LIN {X 0,Y 158.301,Z 763.526,A -85,B 0,C 180,E1 -23831.897,E2 -23831.897} C_VEL
LIN {X 0,Y 156.241,Z 763.233,A -85,B 0,C 180,E1 -23837.005,E2 -23837.005} C_VEL
LIN {X 0,Y 155.491,Z 761.615,A -85,B 0,C 180,E1 -23842.209,E2 -23842.209} C_VEL
LIN {X 0,Y 155.56,Z 760.273,A -85,B 0,C 180,E1 -23844.818,E2 -23844.818} C_VEL
LIN {X 0,Y 155.979,Z 757.524,A -85,B 0,C 180,E1 -23848.711,E2 -23848.711} C_VEL
LIN {X 0,Y 156.074,Z 755.027,A -85,B 0,C 180,E1 -23851.292,E2 -23851.292} C_VEL
LIN {X 0,Y 156.073,Z 750.262,A -85,B 0,C 180,E1 -23855.169,E2 -23855.169} C_VEL
LIN {X 0,Y 156.218,Z 744.142,A -85,B 0,C 180,E1 -23859.06,E2 -23859.06} C_VEL
LIN {X 0,Y 156.866,Z 736.53,A -85,B 0,C 180,E1 -23862.947,E2 -23862.947} C_VEL
LIN {X 0,Y 157.853,Z 728.748,A -85,B 0,C 180,E1 -23866.159,E2 -23866.159} C_VEL
LIN {X 0,Y 159.467,Z 718.303,A -85,B 0,C 180,E1 -23869.638,E2 -23869.638} C_VEL
LIN {X 0,Y 160.165,Z 713.944,A -85,B 0,C 180,E1 -23870.878,E2 -23870.878} C_VEL
LIN {X 0,Y 160.339,Z 710.911,A -85,B 0,C 180,E1 -23871.762,E2 -23871.762} C_VEL
LIN {X 0,Y 159.896,Z 708.03,A -85,B 0,C 180,E1 -23872.707,E2 -23872.707} C_VEL
LIN {X 0,Y 158.002,Z 702.633,A -85,B 0,C 180,E1 -23874.702,E2 -23874.702} C_VEL
LIN {X 0,Y 155.669,Z 695.881,A -85,B 0,C 180,E1 -23877.298,E2 -23877.298} C_VEL
LIN {X 0,Y 155.435,Z 691.449,A -85,B 0,C 180,E1 -23878.779,E2 -23878.779} C_VEL
LIN {X 0,Y 156.41,Z 680.785,A -85,B 0,C 180,E1 -23881.753,E2 -23881.753} C_VEL
LIN {X 0,Y 157.105,Z 669.304,A -85,B 0,C 180,E1 -23884.389,E2 -23884.389} C_VEL
LIN {X 0,Y 157.289,Z 656.551,A -85,B 0,C 180,E1 -23886.771,E2 -23886.771} C_VEL
LIN {X 0,Y 156.753,Z 643.83,A -85,B 0,C 180,E1 -23888.709,E2 -23888.709} C_VEL
LIN {X 0,Y 155.505,Z 632.193,A -85,B 0,C 180,E1 -23890.2,E2 -23890.2} C_VEL
LIN {X 0,Y 154.129,Z 625.609,A -85,B 0,C 180,E1 -23891.054,E2 -23891.054} C_VEL
LIN {X 0,Y 153.301,Z 621.385,A -85,B 0,C 180,E1 -23894.885,E2 -23894.885} C_VEL
LIN {X 0,Y 152.123,Z 615.089,A -85,B 0,C 180,E1 -23900.97,E2 -23900.97} C_VEL
LIN {X 0,Y 151.226,Z 610.219,A -85,B 0,C 180,E1 -23906.103,E2 -23906.103} C_VEL
LIN {X 0,Y 150.323,Z 606.285,A -85,B 0,C 180,E1 -23910.599,E2 -23910.599} C_VEL
LIN {X 0,Y 150.215,Z 605.775,A -85,B 0,C 180,E1 -23911.342,E2 -23911.342} C_VEL
LIN {X 0,Y 150.233,Z 605.772,A -85,B 0,C 180,E1 -23915.099,E2 -23915.099} C_VEL
LIN {X 0,Y 150.374,Z 605.756,A -85,B 0,C 180,E1 -23920.903,E2 -23920.903} C_VEL
LIN {X 0,Y 150.471,Z 605.745,A -85,B 0,C 180,E1 -23926.494,E2 -23926.494} C_VEL
LIN {X 0,Y 150.696,Z 605.716,A -85,B 0,C 180,E1 -23929.248,E2 -23929.248} C_VEL
LIN {X 0,Y 150.769,Z 605.703,A -85,B 0,C 180,E1 -23931.96,E2 -23931.96} C_VEL
LIN {X 0,Y 151.224,Z 605.648,A -85,B 0,C 180,E1 -23939.999,E2 -23939.999} C_VEL
LIN {X 0,Y 150.75,Z 605.699,A -85,B 0,C 180,E1 -23948.039,E2 -23948.039} C_VEL
LIN {X 0,Y 150.62,Z 605.721,A -85,B 0,C 180,E1 -23951.505,E2 -23951.505} C_VEL
LIN {X 0,Y 150.371,Z 605.729,A -85,B 0,C 180,E1 -23956.285,E2 -23956.285} C_VEL
LIN {X 0,Y 150.356,Z 605.756,A -85,B 0,C 180,E1 -23960.791,E2 -23960.791} C_VEL
LIN {X 0,Y 150.249,Z 605.748,A -85,B 0,C 180,E1 -23967.281,E2 -23967.281} C_VEL
LIN {X 0,Y 150.224,Z 605.771,A -85,B 0,C 180,E1 -23972.633,E2 -23972.633} C_VEL
LIN {X 0,Y 150.176,Z 605.777,A -85,B 0,C 180,E1 -23977.471,E2 -23977.471} C_VEL
LIN {X 0,Y 150.153,Z 605.779,A -85,B 0,C 180,E1 -23981.503,E2 -23981.503} C_VEL
LIN {X 0,Y 150.144,Z 605.764,A -85,B 0,C 180,E1 -23985.399,E2 -23985.399} C_VEL
LIN {X 0,Y 150.162,Z 605.778,A -85,B 0,C 180,E1 -23989.06,E2 -23989.06} C_VEL
LIN {X 0,Y 150.218,Z 605.759,A -85,B 0,C 180,E1 -23992.687,E2 -23992.687} C_VEL
LIN {X 0,Y 150.219,Z 605.765,A -85,B 0,C 180,E1 -23997.364,E2 -23997.364} C_VEL
LIN {X 0,Y 150.294,Z 605.761,A -85,B 0,C 180,E1 -24003.948,E2 -24003.948} C_VEL
LIN {X 0,Y 151.357,Z 608.655,A -85,B 0,C 180,E1 -24004.641,E2 -24004.641} C_VEL
LIN {X 0,Y 156.151,Z 618.519,A -85,B 0,C 180,E1 -24007.498,E2 -24007.498} C_VEL
LIN {X 0,Y 159.415,Z 627.15,A -85,B 0,C 180,E1 -24010.001,E2 -24010.001} C_VEL
LIN {X 0,Y 162.002,Z 635.852,A -85,B 0,C 180,E1 -24012.629,E2 -24012.629} C_VEL
LIN {X 0,Y 163.752,Z 643.431,A -85,B 0,C 180,E1 -24015.075,E2 -24015.075} C_VEL
LIN {X 0,Y 161.104,Z 653.934,A -85,B 0,C 180,E1 -24018.039,E2 -24018.039} C_VEL
LIN {X 0,Y 158.728,Z 662.491,A -85,B 0,C 180,E1 -24021.083,E2 -24021.083} C_VEL
LIN {X 0,Y 156.32,Z 670.812,A -85,B 0,C 180,E1 -24024.839,E2 -24024.839} C_VEL
LIN {X 0,Y 154.304,Z 677.372,A -85,B 0,C 180,E1 -24028.562,E2 -24028.562} C_VEL
LIN {X 0,Y 152.679,Z 683.001,A -85,B 0,C 180,E1 -24032.636,E2 -24032.636} C_VEL
LIN {X 0,Y 151.64,Z 687.263,A -85,B 0,C 180,E1 -24036.651,E2 -24036.651} C_VEL
LIN {X 0,Y 151.203,Z 690.46,A -85,B 0,C 180,E1 -24040.712,E2 -24040.712} C_VEL
LIN {X 0,Y 151.19,Z 692.074,A -85,B 0,C 180,E1 -24043.437,E2 -24043.437} C_VEL
LIN {X 0,Y 151.427,Z 693.228,A -85,B 0,C 180,E1 -24046.166,E2 -24046.166} C_VEL
LIN {X 0,Y 152.738,Z 694.356,A -85,B 0,C 180,E1 -24051.596,E2 -24051.596} C_VEL
LIN {X 0,Y 153.787,Z 694.304,A -85,B 0,C 180,E1 -24054.283,E2 -24054.283} C_VEL
LIN {X 0,Y 155.07,Z 693.827,A -85,B 0,C 180,E1 -24056.947,E2 -24056.947} C_VEL
LIN {X 0,Y 156.658,Z 692.946,A -85,B 0,C 180,E1 -24059.567,E2 -24059.567} C_VEL
LIN {X 0,Y 159.152,Z 691.108,A -85,B 0,C 180,E1 -24062.965,E2 -24062.965} C_VEL
LIN {X 0,Y 162.943,Z 687.635,A -85,B 0,C 180,E1 -24067.142,E2 -24067.142} C_VEL
LIN {X 0,Y 166.847,Z 683.387,A -85,B 0,C 180,E1 -24070.696,E2 -24070.696} C_VEL
LIN {X 0,Y 169.613,Z 680.051,A -85,B 0,C 180,E1 -24072.876,E2 -24072.876} C_VEL
LIN {X 0,Y 169.655,Z 678.661,A -85,B 0,C 180,E1 -24074.075,E2 -24074.075} C_VEL
LIN {X 0,Y 160.365,Z 677.774,A -85,B 0,C 180,E1 -24078.901,E2 -24078.901} C_VEL
LIN {X 0,Y 156.701,Z 676.883,A -85,B 0,C 180,E1 -24081.518,E2 -24081.518} C_VEL
LIN {X 0,Y 156.522,Z 676.909,A -85,B 0,C 180,E1 -24081.773,E2 -24081.773} C_VEL
LIN {X 0,Y 154.558,Z 688.668,A -85,B 0,C 180,E1 -24084.33,E2 -24084.33} C_VEL
LIN {X 0,Y 152.548,Z 700.573,A -85,B 0,C 180,E1 -24087.619,E2 -24087.619} C_VEL
LIN {X 0,Y 150.917,Z 709.743,A -85,B 0,C 180,E1 -24090.728,E2 -24090.728} C_VEL
LIN {X 0,Y 149.6,Z 718.707,A -85,B 0,C 180,E1 -24094.423,E2 -24094.423} C_VEL
LIN {X 0,Y 148.6,Z 726.73,A -85,B 0,C 180,E1 -24098.499,E2 -24098.499} C_VEL
LIN {X 0,Y 148.01,Z 733.166,A -85,B 0,C 180,E1 -24102.538,E2 -24102.538} C_VEL
LIN {X 0,Y 147.744,Z 739.641,A -85,B 0,C 180,E1 -24107.641,E2 -24107.641} C_VEL
LIN {X 0,Y 148.22,Z 743.771,A -85,B 0,C 180,E1 -24111.823,E2 -24111.823} C_VEL
LIN {X 0,Y 149.77,Z 747.73,A -85,B 0,C 180,E1 -24117.311,E2 -24117.311} C_VEL
LIN {X 0,Y 152.483,Z 750.261,A -85,B 0,C 180,E1 -24122.643,E2 -24122.643} C_VEL
LIN {X 0,Y 156.515,Z 751.332,A -85,B 0,C 180,E1 -24127.743,E2 -24127.743} C_VEL
LIN {X 0,Y 161.797,Z 751.029,A -85,B 0,C 180,E1 -24132.545,E2 -24132.545} C_VEL
LIN {X 0,Y 168.358,Z 749.378,A -85,B 0,C 180,E1 -24136.991,E2 -24136.991} C_VEL
LIN {X 0,Y 175.968,Z 746.261,A -85,B 0,C 180,E1 -24141.067,E2 -24141.067} C_VEL
LIN {X 0,Y 184.615,Z 741.664,A -85,B 0,C 180,E1 -24144.757,E2 -24144.757} C_VEL
LIN {X 0,Y 194.158,Z 735.354,A -85,B 0,C 180,E1 -24148.072,E2 -24148.072} C_VEL
LIN {X 0,Y 203.161,Z 728.262,A -85,B 0,C 180,E1 -24150.681,E2 -24150.681} C_VEL
LIN {X 0,Y 205.743,Z 726,A -85,B 0,C 180,E1 -24151.357,E2 -24151.357} C_VEL
LIN {X 0,Y 208.061,Z 723.711,A -85,B 0,C 180,E1 -24152.716,E2 -24152.716} C_VEL
LIN {X 0,Y 209.401,Z 722.346,A -85,B 0,C 180,E1 -24153.628,E2 -24153.628} C_VEL
LIN {X 0,Y 210.467,Z 721.212,A -85,B 0,C 180,E1 -24154.589,E2 -24154.589} C_VEL
LIN {X 0,Y 211.809,Z 720.065,A -85,B 0,C 180,E1 -24157.221,E2 -24157.221} C_VEL
LIN {X 0,Y 212.367,Z 720.043,A -85,B 0,C 180,E1 -24158.961,E2 -24158.961} C_VEL
LIN {X 0,Y 209.953,Z 722.891,A -85,B 0,C 180,E1 -24160.353,E2 -24160.353} C_VEL
LIN {X 0,Y 204.984,Z 728.502,A -85,B 0,C 180,E1 -24162.515,E2 -24162.515} C_VEL
LIN {X 0,Y 199.025,Z 734.248,A -85,B 0,C 180,E1 -24164.354,E2 -24164.354} C_VEL
LIN {X 0,Y 190.597,Z 741.609,A -85,B 0,C 180,E1 -24166.99,E2 -24166.99} C_VEL
LIN {X 0,Y 181.392,Z 748.549,A -85,B 0,C 180,E1 -24170.264,E2 -24170.264} C_VEL
LIN {X 0,Y 174.835,Z 752.856,A -85,B 0,C 180,E1 -24172.92,E2 -24172.92} C_VEL
LIN {X 0,Y 167.216,Z 757.285,A -85,B 0,C 180,E1 -24176.884,E2 -24176.884} C_VEL
LIN {X 0,Y 160.578,Z 760.437,A -85,B 0,C 180,E1 -24181.224,E2 -24181.224} C_VEL
LIN {X 0,Y 155.447,Z 762.353,A -85,B 0,C 180,E1 -24185.992,E2 -24185.992} C_VEL
LIN {X 0,Y 151.563,Z 763.014,A -85,B 0,C 180,E1 -24191.062,E2 -24191.062} C_VEL
LIN {X 0,Y 149.342,Z 762.396,A -85,B 0,C 180,E1 -24196.393,E2 -24196.393} C_VEL
LIN {X 0,Y 148.515,Z 760.499,A -85,B 0,C 180,E1 -24201.841,E2 -24201.841} C_VEL
LIN {X 0,Y 148.602,Z 759.026,A -85,B 0,C 180,E1 -24204.575,E2 -24204.575} C_VEL
LIN {X 0,Y 149.043,Z 756.066,A -85,B 0,C 180,E1 -24208.652,E2 -24208.652} C_VEL
LIN {X 0,Y 149.112,Z 753.462,A -85,B 0,C 180,E1 -24211.353,E2 -24211.353} C_VEL
LIN {X 0,Y 149.116,Z 748.437,A -85,B 0,C 180,E1 -24215.411,E2 -24215.411} C_VEL
LIN {X 0,Y 149.329,Z 742.021,A -85,B 0,C 180,E1 -24219.482,E2 -24219.482} C_VEL
LIN {X 0,Y 150.05,Z 733.972,A -85,B 0,C 180,E1 -24223.546,E2 -24223.546} C_VEL
LIN {X 0,Y 151.356,Z 724.046,A -85,B 0,C 180,E1 -24227.569,E2 -24227.569} C_VEL
LIN {X 0,Y 153.223,Z 712.726,A -85,B 0,C 180,E1 -24231.177,E2 -24231.177} C_VEL
LIN {X 0,Y 153.805,Z 709.196,A -85,B 0,C 180,E1 -24232.149,E2 -24232.149} C_VEL
LIN {X 0,Y 154.545,Z 700.824,A -85,B 0,C 180,E1 -24235.597,E2 -24235.597} C_VEL
LIN {X 0,Y 155.435,Z 691.449,A -85,B 0,C 180,E1 -24238.779,E2 -24238.779} C_VEL
LIN {X 0,Y 155.253,Z 686.965,A -85,B 0,C 180,E1 -24240.18,E2 -24240.18} C_VEL
LIN {X 0,Y 153.152,Z 679.582,A -85,B 0,C 180,E1 -24242.533,E2 -24242.533} C_VEL
LIN {X 0,Y 151.003,Z 671.94,A -85,B 0,C 180,E1 -24244.804,E2 -24244.804} C_VEL
LIN {X 0,Y 150.63,Z 666.943,A -85,B 0,C 180,E1 -24246.014,E2 -24246.014} C_VEL
LIN {X 0,Y 150.901,Z 653.621,A -85,B 0,C 180,E1 -24248.535,E2 -24248.535} C_VEL
LIN {X 0,Y 150.259,Z 639.839,A -85,B 0,C 180,E1 -24250.68,E2 -24250.68} C_VEL
LIN {X 0,Y 148.895,Z 630.887,A -85,B 0,C 180,E1 -24251.953,E2 -24251.953} C_VEL
LIN {X 0,Y 148.126,Z 628.352,A -85,B 0,C 180,E1 -24252.388,E2 -24252.388} C_VEL
LIN {X 0,Y 146.693,Z 624.312,A -85,B 0,C 180,E1 -24253.127,E2 -24253.127} C_VEL
LIN {X 0,Y 145.429,Z 618.159,A -85,B 0,C 180,E1 -24259.278,E2 -24259.278} C_VEL
LIN {X 0,Y 144.594,Z 613.43,A -85,B 0,C 180,E1 -24264.318,E2 -24264.318} C_VEL
LIN {X 0,Y 143.805,Z 609.245,A -85,B 0,C 180,E1 -24269.125,E2 -24269.125} C_VEL
LIN {X 0,Y 143.216,Z 606.645,A -85,B 0,C 180,E1 -24272.488,E2 -24272.488} C_VEL
LIN {X 0,Y 143.284,Z 606.64,A -85,B 0,C 180,E1 -24278.745,E2 -24278.745} C_VEL
LIN {X 0,Y 143.323,Z 606.636,A -85,B 0,C 180,E1 -24282.888,E2 -24282.888} C_VEL
LIN {X 0,Y 143.609,Z 606.598,A -85,B 0,C 180,E1 -24288.71,E2 -24288.71} C_VEL
LIN {X 0,Y 143.691,Z 606.585,A -85,B 0,C 180,E1 -24291.561,E2 -24291.561} C_VEL
LIN {X 0,Y 144.183,Z 606.525,A -85,B 0,C 180,E1 -24299.999,E2 -24299.999} C_VEL
LIN {X 0,Y 143.671,Z 606.583,A -85,B 0,C 180,E1 -24308.438,E2 -24308.438} C_VEL
LIN {X 0,Y 143.553,Z 606.602,A -85,B 0,C 180,E1 -24311.711,E2 -24311.711} C_VEL
LIN {X 0,Y 143.309,Z 606.611,A -85,B 0,C 180,E1 -24317.111,E2 -24317.111} C_VEL
LIN {X 0,Y 143.282,Z 606.637,A -85,B 0,C 180,E1 -24321.253,E2 -24321.253} C_VEL
LIN {X 0,Y 143.196,Z 606.629,A -85,B 0,C 180,E1 -24327.936,E2 -24327.936} C_VEL
LIN {X 0,Y 143.151,Z 606.65,A -85,B 0,C 180,E1 -24333.42,E2 -24333.42} C_VEL
LIN {X 0,Y 143.064,Z 606.661,A -85,B 0,C 180,E1 -24339.688,E2 -24339.688} C_VEL
LIN {X 0,Y 143.064,Z 606.651,A -85,B 0,C 180,E1 -24343.451,E2 -24343.451} C_VEL
LIN {X 0,Y 143.075,Z 606.658,A -85,B 0,C 180,E1 -24347.459,E2 -24347.459} C_VEL
LIN {X 0,Y 143.11,Z 606.644,A -85,B 0,C 180,E1 -24351.788,E2 -24351.788} C_VEL
LIN {X 0,Y 143.187,Z 606.641,A -85,B 0,C 180,E1 -24357.32,E2 -24357.32} C_VEL
LIN {X 0,Y 143.193,Z 606.812,A -85,B 0,C 180,E1 -24361.958,E2 -24361.958} C_VEL
LIN {X 0,Y 144.278,Z 609.57,A -85,B 0,C 180,E1 -24362.706,E2 -24362.706} C_VEL
LIN {X 0,Y 145.183,Z 610.769,A -85,B 0,C 180,E1 -24363.162,E2 -24363.162} C_VEL
LIN {X 0,Y 150.317,Z 621.884,A -85,B 0,C 180,E1 -24366.646,E2 -24366.646} C_VEL
LIN {X 0,Y 153.24,Z 629.925,A -85,B 0,C 180,E1 -24369.159,E2 -24369.159} C_VEL
LIN {X 0,Y 155.662,Z 638.385,A -85,B 0,C 180,E1 -24371.911,E2 -24371.911} C_VEL
LIN {X 0,Y 157.084,Z 644.663,A -85,B 0,C 180,E1 -24374.091,E2 -24374.091} C_VEL
LIN {X 0,Y 156.799,Z 646.889,A -85,B 0,C 180,E1 -24374.73,E2 -24374.73} C_VEL
LIN {X 0,Y 154.248,Z 656.012,A -85,B 0,C 180,E1 -24377.499,E2 -24377.499} C_VEL
LIN {X 0,Y 151.293,Z 665.84,A -85,B 0,C 180,E1 -24381.314,E2 -24381.314} C_VEL
LIN {X 0,Y 149.248,Z 672.533,A -85,B 0,C 180,E1 -24384.593,E2 -24384.593} C_VEL
LIN {X 0,Y 147.198,Z 678.965,A -85,B 0,C 180,E1 -24388.493,E2 -24388.493} C_VEL
LIN {X 0,Y 145.543,Z 684.488,A -85,B 0,C 180,E1 -24392.765,E2 -24392.765} C_VEL
LIN {X 0,Y 144.535,Z 688.645,A -85,B 0,C 180,E1 -24396.98,E2 -24396.98} C_VEL
LIN {X 0,Y 144.119,Z 692.599,A -85,B 0,C 180,E1 -24402.765,E2 -24402.765} C_VEL
LIN {X 0,Y 144.507,Z 694.378,A -85,B 0,C 180,E1 -24406.963,E2 -24406.963} C_VEL
LIN {X 0,Y 145.122,Z 695.092,A -85,B 0,C 180,E1 -24409.813,E2 -24409.813} C_VEL
LIN {X 0,Y 146.778,Z 695.372,A -85,B 0,C 180,E1 -24414.531,E2 -24414.531} C_VEL
LIN {X 0,Y 148.63,Z 694.749,A -85,B 0,C 180,E1 -24418.217,E2 -24418.217} C_VEL
LIN {X 0,Y 150.388,Z 693.823,A -85,B 0,C 180,E1 -24420.931,E2 -24420.931} C_VEL
LIN {X 0,Y 152.794,Z 692.109,A -85,B 0,C 180,E1 -24424.114,E2 -24424.114} C_VEL
LIN {X 0,Y 157.18,Z 688.318,A -85,B 0,C 180,E1 -24428.751,E2 -24428.751} C_VEL
LIN {X 0,Y 161.717,Z 683.57,A -85,B 0,C 180,E1 -24432.653,E2 -24432.653} C_VEL
LIN {X 0,Y 162.855,Z 682.122,A -85,B 0,C 180,E1 -24433.665,E2 -24433.665} C_VEL
LIN {X 0,Y 148.855,Z 680.705,A -85,B 0,C 180,E1 -24442.138,E2 -24442.138} C_VEL
LIN {X 0,Y 148.753,Z 680.967,A -85,B 0,C 180,E1 -24442.302,E2 -24442.302} C_VEL
LIN {X 0,Y 146.676,Z 693.215,A -85,B 0,C 180,E1 -24445.321,E2 -24445.321} C_VEL
LIN {X 0,Y 144.857,Z 703.701,A -85,B 0,C 180,E1 -24448.565,E2 -24448.565} C_VEL
LIN {X 0,Y 143.193,Z 713.525,A -85,B 0,C 180,E1 -24452.326,E2 -24452.326} C_VEL
LIN {X 0,Y 141.938,Z 722.688,A -85,B 0,C 180,E1 -24456.666,E2 -24456.666} C_VEL
LIN {X 0,Y 141.116,Z 730.253,A -85,B 0,C 180,E1 -24461.121,E2 -24461.121} C_VEL
LIN {X 0,Y 140.701,Z 736.342,A -85,B 0,C 180,E1 -24465.538,E2 -24465.538} C_VEL
LIN {X 0,Y 140.859,Z 741.194,A -85,B 0,C 180,E1 -24469.944,E2 -24469.944} C_VEL
LIN {X 0,Y 141.708,Z 745.045,A -85,B 0,C 180,E1 -24474.309,E2 -24474.309} C_VEL
LIN {X 0,Y 143.696,Z 748.787,A -85,B 0,C 180,E1 -24480.001,E2 -24480.001} C_VEL
LIN {X 0,Y 147.161,Z 751.048,A -85,B 0,C 180,E1 -24485.482,E2 -24485.482} C_VEL
LIN {X 0,Y 151.908,Z 751.944,A -85,B 0,C 180,E1 -24490.666,E2 -24490.666} C_VEL
LIN {X 0,Y 157.986,Z 751.504,A -85,B 0,C 180,E1 -24495.481,E2 -24495.481} C_VEL
LIN {X 0,Y 165.278,Z 749.664,A -85,B 0,C 180,E1 -24499.889,E2 -24499.889} C_VEL
LIN {X 0,Y 173.654,Z 746.42,A -85,B 0,C 180,E1 -24503.874,E2 -24503.874} C_VEL
LIN {X 0,Y 183.018,Z 741.682,A -85,B 0,C 180,E1 -24507.44,E2 -24507.44} C_VEL
LIN {X 0,Y 193.229,Z 735.201,A -85,B 0,C 180,E1 -24510.611,E2 -24510.611} C_VEL
LIN {X 0,Y 201.391,Z 729.127,A -85,B 0,C 180,E1 -24512.745,E2 -24512.745} C_VEL
LIN {X 0,Y 204.235,Z 726.638,A -85,B 0,C 180,E1 -24514.327,E2 -24514.327} C_VEL
LIN {X 0,Y 205.566,Z 725.568,A -85,B 0,C 180,E1 -24515.536,E2 -24515.536} C_VEL
LIN {X 0,Y 206.692,Z 724.829,A -85,B 0,C 180,E1 -24517.738,E2 -24517.738} C_VEL
LIN {X 0,Y 206.7,Z 725.081,A -85,B 0,C 180,E1 -24518.557,E2 -24518.557} C_VEL
LIN {X 0,Y 202.724,Z 729.061,A -85,B 0,C 180,E1 -24520.301,E2 -24520.301} C_VEL
LIN {X 0,Y 199.389,Z 732.222,A -85,B 0,C 180,E1 -24521.498,E2 -24521.498} C_VEL
LIN {X 0,Y 190.514,Z 739.613,A -85,B 0,C 180,E1 -24524.002,E2 -24524.002} C_VEL
LIN {X 0,Y 180.858,Z 746.721,A -85,B 0,C 180,E1 -24527.157,E2 -24527.157} C_VEL
LIN {X 0,Y 171.462,Z 752.467,A -85,B 0,C 180,E1 -24530.559,E2 -24530.559} C_VEL
LIN {X 0,Y 165.169,Z 755.88,A -85,B 0,C 180,E1 -24533.44,E2 -24533.44} C_VEL
LIN {X 0,Y 157.666,Z 759.265,A -85,B 0,C 180,E1 -24537.666,E2 -24537.666} C_VEL
LIN {X 0,Y 151.555,Z 761.417,A -85,B 0,C 180,E1 -24542.375,E2 -24542.375} C_VEL
LIN {X 0,Y 146.794,Z 762.358,A -85,B 0,C 180,E1 -24547.482,E2 -24547.482} C_VEL
LIN {X 0,Y 143.448,Z 762.076,A -85,B 0,C 180,E1 -24552.908,E2 -24552.908} C_VEL
LIN {X 0,Y 141.816,Z 760.568,A -85,B 0,C 180,E1 -24558.569,E2 -24558.569} C_VEL
LIN {X 0,Y 141.655,Z 757.737,A -85,B 0,C 180,E1 -24564.308,E2 -24564.308} C_VEL
LIN {X 0,Y 142.121,Z 754.561,A -85,B 0,C 180,E1 -24568.586,E2 -24568.586} C_VEL
LIN {X 0,Y 142.183,Z 751.749,A -85,B 0,C 180,E1 -24571.419,E2 -24571.419} C_VEL
LIN {X 0,Y 142.16,Z 746.462,A -85,B 0,C 180,E1 -24575.677,E2 -24575.677} C_VEL
LIN {X 0,Y 142.412,Z 739.746,A -85,B 0,C 180,E1 -24579.947,E2 -24579.947} C_VEL
LIN {X 0,Y 143.232,Z 731.342,A -85,B 0,C 180,E1 -24584.204,E2 -24584.204} C_VEL
LIN {X 0,Y 144.669,Z 720.828,A -85,B 0,C 180,E1 -24588.41,E2 -24588.41} C_VEL
LIN {X 0,Y 146.443,Z 710.42,A -85,B 0,C 180,E1 -24591.837,E2 -24591.837} C_VEL
LIN {X 0,Y 147.102,Z 706.091,A -85,B 0,C 180,E1 -24593.883,E2 -24593.883} C_VEL
LIN {X 0,Y 147.974,Z 697.037,A -85,B 0,C 180,E1 -24597.588,E2 -24597.588} C_VEL
LIN {X 0,Y 149.049,Z 687.304,A -85,B 0,C 180,E1 -24600.852,E2 -24600.852} C_VEL
LIN {X 0,Y 150.078,Z 676.231,A -85,B 0,C 180,E1 -24603.88,E2 -24603.88} C_VEL
LIN {X 0,Y 150.63,Z 666.943,A -85,B 0,C 180,E1 -24606.014,E2 -24606.014} C_VEL
LIN {X 0,Y 150.216,Z 661.901,A -85,B 0,C 180,E1 -24607.18,E2 -24607.18} C_VEL
LIN {X 0,Y 147.668,Z 653.919,A -85,B 0,C 180,E1 -24609.236,E2 -24609.236} C_VEL
LIN {X 0,Y 144.9,Z 645.742,A -85,B 0,C 180,E1 -24611.2,E2 -24611.2} C_VEL
LIN {X 0,Y 144.081,Z 640.381,A -85,B 0,C 180,E1 -24612.168,E2 -24612.168} C_VEL
LIN {X 0,Y 142.976,Z 632.465,A -85,B 0,C 180,E1 -24613.424,E2 -24613.424} C_VEL
LIN {X 0,Y 140.902,Z 627.616,A -85,B 0,C 180,E1 -24614.503,E2 -24614.503} C_VEL
LIN {X 0,Y 139.436,Z 624.264,A -85,B 0,C 180,E1 -24615.233,E2 -24615.233} C_VEL
LIN {X 0,Y 139.138,Z 623.031,A -85,B 0,C 180,E1 -24615.504,E2 -24615.504} C_VEL
LIN {X 0,Y 138.198,Z 617.877,A -85,B 0,C 180,E1 -24620.98,E2 -24620.98} C_VEL
LIN {X 0,Y 137.446,Z 613.695,A -85,B 0,C 180,E1 -24625.772,E2 -24625.772} C_VEL
LIN {X 0,Y 136.912,Z 610.962,A -85,B 0,C 180,E1 -24629.113,E2 -24629.113} C_VEL
LIN {X 0,Y 136.135,Z 607.528,A -85,B 0,C 180,E1 -24633.764,E2 -24633.764} C_VEL
LIN {X 0,Y 136.251,Z 607.517,A -85,B 0,C 180,E1 -24638.833,E2 -24638.833} C_VEL
LIN {X 0,Y 136.292,Z 607.512,A -85,B 0,C 180,E1 -24645.058,E2 -24645.058} C_VEL
LIN {X 0,Y 136.508,Z 607.481,A -85,B 0,C 180,E1 -24648.114,E2 -24648.114} C_VEL
LIN {X 0,Y 136.615,Z 607.468,A -85,B 0,C 180,E1 -24651.121,E2 -24651.121} C_VEL
LIN {X 0,Y 137.14,Z 607.402,A -85,B 0,C 180,E1 -24659.999,E2 -24659.999} C_VEL
LIN {X 0,Y 136.598,Z 607.466,A -85,B 0,C 180,E1 -24668.878,E2 -24668.878} C_VEL
LIN {X 0,Y 136.497,Z 607.479,A -85,B 0,C 180,E1 -24671.953,E2 -24671.953} C_VEL
LIN {X 0,Y 136.249,Z 607.496,A -85,B 0,C 180,E1 -24678.027,E2 -24678.027} C_VEL
LIN {X 0,Y 136.203,Z 607.519,A -85,B 0,C 180,E1 -24681.747,E2 -24681.747} C_VEL
LIN {X 0,Y 136.122,Z 607.514,A -85,B 0,C 180,E1 -24688.628,E2 -24688.628} C_VEL
LIN {X 0,Y 136.048,Z 607.534,A -85,B 0,C 180,E1 -24694.626,E2 -24694.626} C_VEL
LIN {X 0,Y 136.034,Z 607.535,A -85,B 0,C 180,E1 -24699.196,E2 -24699.196} C_VEL
LIN {X 0,Y 136.005,Z 607.528,A -85,B 0,C 180,E1 -24703.657,E2 -24703.657} C_VEL
LIN {X 0,Y 136.038,Z 607.535,A -85,B 0,C 180,E1 -24707.806,E2 -24707.806} C_VEL
LIN {X 0,Y 136.059,Z 607.522,A -85,B 0,C 180,E1 -24711.692,E2 -24711.692} C_VEL
LIN {X 0,Y 136.092,Z 607.532,A -85,B 0,C 180,E1 -24715.715,E2 -24715.715} C_VEL
LIN {X 0,Y 136.084,Z 607.644,A -85,B 0,C 180,E1 -24719.661,E2 -24719.661} C_VEL
LIN {X 0,Y 137.091,Z 610.383,A -85,B 0,C 180,E1 -24720.456,E2 -24720.456} C_VEL
LIN {X 0,Y 140.441,Z 616.118,A -85,B 0,C 180,E1 -24722.591,E2 -24722.591} C_VEL
LIN {X 0,Y 144.604,Z 625.56,A -85,B 0,C 180,E1 -24725.832,E2 -24725.832} C_VEL
LIN {X 0,Y 147.586,Z 634.312,A -85,B 0,C 180,E1 -24728.832,E2 -24728.832} C_VEL
LIN {X 0,Y 149.727,Z 642.745,A -85,B 0,C 180,E1 -24731.825,E2 -24731.825} C_VEL
LIN {X 0,Y 150.595,Z 646.913,A -85,B 0,C 180,E1 -24733.386,E2 -24733.386} C_VEL
LIN {X 0,Y 147.916,Z 656.228,A -85,B 0,C 180,E1 -24736.255,E2 -24736.255} C_VEL
LIN {X 0,Y 145.289,Z 664.727,A -85,B 0,C 180,E1 -24739.546,E2 -24739.546} C_VEL
LIN {X 0,Y 142.6,Z 673.013,A -85,B 0,C 180,E1 -24743.631,E2 -24743.631} C_VEL
LIN {X 0,Y 140.354,Z 679.742,A -85,B 0,C 180,E1 -24747.845,E2 -24747.845} C_VEL
LIN {X 0,Y 138.394,Z 685.947,A -85,B 0,C 180,E1 -24752.908,E2 -24752.908} C_VEL
LIN {X 0,Y 137.44,Z 689.992,A -85,B 0,C 180,E1 -24757.342,E2 -24757.342} C_VEL
LIN {X 0,Y 137.089,Z 693.663,A -85,B 0,C 180,E1 -24763.087,E2 -24763.087} C_VEL
LIN {X 0,Y 137.614,Z 695.528,A -85,B 0,C 180,E1 -24767.841,E2 -24767.841} C_VEL
LIN {X 0,Y 138.336,Z 696.197,A -85,B 0,C 180,E1 -24770.829,E2 -24770.829} C_VEL
LIN {X 0,Y 140.04,Z 696.395,A -85,B 0,C 180,E1 -24775.402,E2 -24775.402} C_VEL
LIN {X 0,Y 142.271,Z 695.674,A -85,B 0,C 180,E1 -24779.6,E2 -24779.6} C_VEL
LIN {X 0,Y 144.183,Z 694.68,A -85,B 0,C 180,E1 -24782.42,E2 -24782.42} C_VEL
LIN {X 0,Y 146.535,Z 693.096,A -85,B 0,C 180,E1 -24785.381,E2 -24785.381} C_VEL
LIN {X 0,Y 150.163,Z 690.2,A -85,B 0,C 180,E1 -24789.182,E2 -24789.182} C_VEL
LIN {X 0,Y 155.275,Z 685.304,A -85,B 0,C 180,E1 -24793.601,E2 -24793.601} C_VEL
LIN {X 0,Y 144.04,Z 684.497,A -85,B 0,C 180,E1 -24800.634,E2 -24800.634} C_VEL
LIN {X 0,Y 141.905,Z 684.676,A -85,B 0,C 180,E1 -24801.755,E2 -24801.755} C_VEL
LIN {X 0,Y 141.096,Z 684.436,A -85,B 0,C 180,E1 -24802.804,E2 -24802.804} C_VEL
LIN {X 0,Y 138.98,Z 696.61,A -85,B 0,C 180,E1 -24806.204,E2 -24806.204} C_VEL
LIN {X 0,Y 137.088,Z 706.873,A -85,B 0,C 180,E1 -24809.768,E2 -24809.768} C_VEL
LIN {X 0,Y 135.638,Z 716.443,A -85,B 0,C 180,E1 -24813.871,E2 -24813.871} C_VEL
LIN {X 0,Y 134.49,Z 725.292,A -85,B 0,C 180,E1 -24818.545,E2 -24818.545} C_VEL
LIN {X 0,Y 133.863,Z 732.394,A -85,B 0,C 180,E1 -24823.218,E2 -24823.218} C_VEL
LIN {X 0,Y 133.673,Z 738.074,A -85,B 0,C 180,E1 -24827.861,E2 -24827.861} C_VEL
LIN {X 0,Y 134.517,Z 743.974,A -85,B 0,C 180,E1 -24834.003,E2 -24834.003} C_VEL
LIN {X 0,Y 136.485,Z 748.19,A -85,B 0,C 180,E1 -24840.001,E2 -24840.001} C_VEL
LIN {X 0,Y 139.963,Z 750.948,A -85,B 0,C 180,E1 -24845.765,E2 -24845.765} C_VEL
LIN {X 0,Y 144.81,Z 752.354,A -85,B 0,C 180,E1 -24851.195,E2 -24851.195} C_VEL
LIN {X 0,Y 151.072,Z 752.429,A -85,B 0,C 180,E1 -24856.209,E2 -24856.209} C_VEL
LIN {X 0,Y 158.573,Z 751.131,A -85,B 0,C 180,E1 -24860.768,E2 -24860.768} C_VEL
LIN {X 0,Y 167.186,Z 748.485,A -85,B 0,C 180,E1 -24864.859,E2 -24864.859} C_VEL
LIN {X 0,Y 176.772,Z 744.391,A -85,B 0,C 180,E1 -24868.497,E2 -24868.497} C_VEL
LIN {X 0,Y 187.272,Z 738.671,A -85,B 0,C 180,E1 -24871.696,E2 -24871.696} C_VEL
LIN {X 0,Y 195.29,Z 733.406,A -85,B 0,C 180,E1 -24873.771,E2 -24873.771} C_VEL
LIN {X 0,Y 198.065,Z 731.426,A -85,B 0,C 180,E1 -24874.593,E2 -24874.593} C_VEL
LIN {X 0,Y 200.307,Z 729.872,A -85,B 0,C 180,E1 -24876.202,E2 -24876.202} C_VEL
LIN {X 0,Y 200.488,Z 729.775,A -85,B 0,C 180,E1 -24876.58,E2 -24876.58} C_VEL
LIN {X 0,Y 200.502,Z 730.053,A -85,B 0,C 180,E1 -24878.097,E2 -24878.097} C_VEL
LIN {X 0,Y 196.281,Z 733.704,A -85,B 0,C 180,E1 -24879.665,E2 -24879.665} C_VEL
LIN {X 0,Y 185.812,Z 741.561,A -85,B 0,C 180,E1 -24882.48,E2 -24882.48} C_VEL
LIN {X 0,Y 175.8,Z 748.064,A -85,B 0,C 180,E1 -24885.608,E2 -24885.608} C_VEL
LIN {X 0,Y 166.1,Z 753.373,A -85,B 0,C 180,E1 -24889.02,E2 -24889.02} C_VEL
LIN {X 0,Y 159.544,Z 756.397,A -85,B 0,C 180,E1 -24891.927,E2 -24891.927} C_VEL
LIN {X 0,Y 151.716,Z 759.409,A -85,B 0,C 180,E1 -24896.232,E2 -24896.232} C_VEL
LIN {X 0,Y 145.278,Z 761.216,A -85,B 0,C 180,E1 -24901.072,E2 -24901.072} C_VEL
LIN {X 0,Y 140.262,Z 761.823,A -85,B 0,C 180,E1 -24906.372,E2 -24906.372} C_VEL
LIN {X 0,Y 136.706,Z 761.207,A -85,B 0,C 180,E1 -24912.037,E2 -24912.037} C_VEL
LIN {X 0,Y 134.921,Z 759.41,A -85,B 0,C 180,E1 -24917.977,E2 -24917.977} C_VEL
LIN {X 0,Y 134.716,Z 756.283,A -85,B 0,C 180,E1 -24924.014,E2 -24924.014} C_VEL
LIN {X 0,Y 135.223,Z 752.931,A -85,B 0,C 180,E1 -24928.514,E2 -24928.514} C_VEL
LIN {X 0,Y 135.244,Z 749.965,A -85,B 0,C 180,E1 -24931.492,E2 -24931.492} C_VEL
LIN {X 0,Y 135.215,Z 744.365,A -85,B 0,C 180,E1 -24935.97,E2 -24935.97} C_VEL
LIN {X 0,Y 135.492,Z 737.534,A -85,B 0,C 180,E1 -24940.311,E2 -24940.311} C_VEL
LIN {X 0,Y 136.419,Z 728.462,A -85,B 0,C 180,E1 -24944.93,E2 -24944.93} C_VEL
LIN {X 0,Y 137.698,Z 719.529,A -85,B 0,C 180,E1 -24948.605,E2 -24948.605} C_VEL
LIN {X 0,Y 138.968,Z 712.174,A -85,B 0,C 180,E1 -24951.123,E2 -24951.123} C_VEL
LIN {X 0,Y 140.001,Z 707.36,A -85,B 0,C 180,E1 -24953.681,E2 -24953.681} C_VEL
LIN {X 0,Y 140.829,Z 698.981,A -85,B 0,C 180,E1 -24957.494,E2 -24957.494} C_VEL
LIN {X 0,Y 142.116,Z 688.696,A -85,B 0,C 180,E1 -24961.285,E2 -24961.285} C_VEL
LIN {X 0,Y 143.418,Z 677.065,A -85,B 0,C 180,E1 -24964.759,E2 -24964.759} C_VEL
LIN {X 0,Y 144.186,Z 666.571,A -85,B 0,C 180,E1 -24967.34,E2 -24967.34} C_VEL
LIN {X 0,Y 144.607,Z 653.809,A -85,B 0,C 180,E1 -24969.907,E2 -24969.907} C_VEL
LIN {X 0,Y 144.081,Z 640.381,A -85,B 0,C 180,E1 -24972.168,E2 -24972.168} C_VEL
LIN {X 0,Y 143.19,Z 637.035,A -85,B 0,C 180,E1 -24972.854,E2 -24972.854} C_VEL
LIN {X 0,Y 141.323,Z 634.287,A -85,B 0,C 180,E1 -24973.717,E2 -24973.717} C_VEL
LIN {X 0,Y 134.057,Z 627.235,A -85,B 0,C 180,E1 -24976.741,E2 -24976.741} C_VEL
LIN {X 0,Y 133.391,Z 626.284,A -85,B 0,C 180,E1 -24977.072,E2 -24977.072} C_VEL
LIN {X 0,Y 131.883,Z 622.815,A -85,B 0,C 180,E1 -24977.928,E2 -24977.928} C_VEL
LIN {X 0,Y 131.627,Z 621.631,A -85,B 0,C 180,E1 -24978.245,E2 -24978.245} C_VEL
LIN {X 0,Y 130.838,Z 616.899,A -85,B 0,C 180,E1 -24983.78,E2 -24983.78} C_VEL
LIN {X 0,Y 130.049,Z 612.749,A -85,B 0,C 180,E1 -24988.984,E2 -24988.984} C_VEL
LIN {X 0,Y 129.067,Z 608.409,A -85,B 0,C 180,E1 -24995.145,E2 -24995.145} C_VEL
LIN {X 0,Y 129.167,Z 608.397,A -85,B 0,C 180,E1 -25000.945,E2 -25000.945} C_VEL
LIN {X 0,Y 129.425,Z 608.363,A -85,B 0,C 180,E1 -25007.815,E2 -25007.815} C_VEL
LIN {X 0,Y 129.537,Z 608.351,A -85,B 0,C 180,E1 -25010.631,E2 -25010.631} C_VEL
LIN {X 0,Y 130.095,Z 608.279,A -85,B 0,C 180,E1 -25019.999,E2 -25019.999} C_VEL
LIN {X 0,Y 129.523,Z 608.349,A -85,B 0,C 180,E1 -25029.367,E2 -25029.367} C_VEL
LIN {X 0,Y 129.398,Z 608.359,A -85,B 0,C 180,E1 -25032.546,E2 -25032.546} C_VEL
LIN {X 0,Y 129.16,Z 608.386,A -85,B 0,C 180,E1 -25039.054,E2 -25039.054} C_VEL
LIN {X 0,Y 129.113,Z 608.401,A -85,B 0,C 180,E1 -25042.396,E2 -25042.396} C_VEL
LIN {X 0,Y 129.04,Z 608.401,A -85,B 0,C 180,E1 -25049.371,E2 -25049.371} C_VEL
LIN {X 0,Y 128.964,Z 608.419,A -85,B 0,C 180,E1 -25055.166,E2 -25055.166} C_VEL
LIN {X 0,Y 128.947,Z 608.422,A -85,B 0,C 180,E1 -25060.845,E2 -25060.845} C_VEL
LIN {X 0,Y 128.928,Z 608.405,A -85,B 0,C 180,E1 -25065.123,E2 -25065.123} C_VEL
LIN {X 0,Y 128.984,Z 608.414,A -85,B 0,C 180,E1 -25069.712,E2 -25069.712} C_VEL
LIN {X 0,Y 128.994,Z 608.415,A -85,B 0,C 180,E1 -25074.808,E2 -25074.808} C_VEL
LIN {X 0,Y 129.012,Z 608.497,A -85,B 0,C 180,E1 -25077.063,E2 -25077.063} C_VEL
LIN {X 0,Y 129.97,Z 611.191,A -85,B 0,C 180,E1 -25077.926,E2 -25077.926} C_VEL
LIN {X 0,Y 131.399,Z 613.232,A -85,B 0,C 180,E1 -25078.843,E2 -25078.843} C_VEL
LIN {X 0,Y 135.884,Z 621.939,A -85,B 0,C 180,E1 -25082.256,E2 -25082.256} C_VEL
LIN {X 0,Y 139.694,Z 631.464,A -85,B 0,C 180,E1 -25085.826,E2 -25085.826} C_VEL
LIN {X 0,Y 142.302,Z 640.294,A -85,B 0,C 180,E1 -25089.141,E2 -25089.141} C_VEL
LIN {X 0,Y 143.911,Z 647.899,A -85,B 0,C 180,E1 -25092.122,E2 -25092.122} C_VEL
LIN {X 0,Y 143.957,Z 649.074,A -85,B 0,C 180,E1 -25092.547,E2 -25092.547} C_VEL
LIN {X 0,Y 141.092,Z 658.286,A -85,B 0,C 180,E1 -25095.576,E2 -25095.576} C_VEL
LIN {X 0,Y 138.335,Z 666.589,A -85,B 0,C 180,E1 -25099.014,E2 -25099.014} C_VEL
LIN {X 0,Y 135.56,Z 674.732,A -85,B 0,C 180,E1 -25103.299,E2 -25103.299} C_VEL
LIN {X 0,Y 133.581,Z 680.319,A -85,B 0,C 180,E1 -25106.981,E2 -25106.981} C_VEL
LIN {X 0,Y 131.745,Z 685.81,A -85,B 0,C 180,E1 -25111.526,E2 -25111.526} C_VEL
LIN {X 0,Y 130.571,Z 690.126,A -85,B 0,C 180,E1 -25116.177,E2 -25116.177} C_VEL
LIN {X 0,Y 130.146,Z 692.438,A -85,B 0,C 180,E1 -25119.32,E2 -25119.32} C_VEL
LIN {X 0,Y 130.077,Z 694.737,A -85,B 0,C 180,E1 -25123.465,E2 -25123.465} C_VEL
LIN {X 0,Y 130.775,Z 696.678,A -85,B 0,C 180,E1 -25128.808,E2 -25128.808} C_VEL
LIN {X 0,Y 131.589,Z 697.272,A -85,B 0,C 180,E1 -25131.951,E2 -25131.951} C_VEL
LIN {X 0,Y 134.213,Z 697.216,A -85,B 0,C 180,E1 -25138.114,E2 -25138.114} C_VEL
LIN {X 0,Y 136,Z 696.595,A -85,B 0,C 180,E1 -25141.112,E2 -25141.112} C_VEL
LIN {X 0,Y 140.344,Z 694.087,A -85,B 0,C 180,E1 -25146.754,E2 -25146.754} C_VEL
LIN {X 0,Y 144.57,Z 690.883,A -85,B 0,C 180,E1 -25151.013,E2 -25151.013} C_VEL
LIN {X 0,Y 146.066,Z 689.601,A -85,B 0,C 180,E1 -25152.343,E2 -25152.343} C_VEL
LIN {X 0,Y 146.665,Z 688.289,A -85,B 0,C 180,E1 -25154.048,E2 -25154.048} C_VEL
LIN {X 0,Y 139.208,Z 687.938,A -85,B 0,C 180,E1 -25158.982,E2 -25158.982} C_VEL
LIN {X 0,Y 136.323,Z 688.103,A -85,B 0,C 180,E1 -25160.647,E2 -25160.647} C_VEL
LIN {X 0,Y 133.709,Z 687.921,A -85,B 0,C 180,E1 -25162.823,E2 -25162.823} C_VEL
LIN {X 0,Y 133.417,Z 687.69,A -85,B 0,C 180,E1 -25163.432,E2 -25163.432} C_VEL
LIN {X 0,Y 131.258,Z 699.683,A -85,B 0,C 180,E1 -25167.173,E2 -25167.173} C_VEL
LIN {X 0,Y 129.264,Z 710.952,A -85,B 0,C 180,E1 -25171.594,E2 -25171.594} C_VEL
LIN {X 0,Y 128.069,Z 719.396,A -85,B 0,C 180,E1 -25175.698,E2 -25175.698} C_VEL
LIN {X 0,Y 127.151,Z 727.618,A -85,B 0,C 180,E1 -25180.633,E2 -25180.633} C_VEL
LIN {X 0,Y 126.652,Z 734.258,A -85,B 0,C 180,E1 -25185.541,E2 -25185.541} C_VEL
LIN {X 0,Y 126.804,Z 739.66,A -85,B 0,C 180,E1 -25190.43,E2 -25190.43} C_VEL
LIN {X 0,Y 128.172,Z 745.231,A -85,B 0,C 180,E1 -25196.858,E2 -25196.858} C_VEL
LIN {X 0,Y 130.843,Z 749.191,A -85,B 0,C 180,E1 -25203.08,E2 -25203.08} C_VEL
LIN {X 0,Y 135.242,Z 751.824,A -85,B 0,C 180,E1 -25209.141,E2 -25209.141} C_VEL
LIN {X 0,Y 140.743,Z 753.038,A -85,B 0,C 180,E1 -25214.459,E2 -25214.459} C_VEL
LIN {X 0,Y 147.874,Z 752.94,A -85,B 0,C 180,E1 -25219.433,E2 -25219.433} C_VEL
LIN {X 0,Y 156.145,Z 751.544,A -85,B 0,C 180,E1 -25223.898,E2 -25223.898} C_VEL
LIN {X 0,Y 165.557,Z 748.793,A -85,B 0,C 180,E1 -25227.838,E2 -25227.838} C_VEL
LIN {X 0,Y 175.847,Z 744.583,A -85,B 0,C 180,E1 -25231.304,E2 -25231.304} C_VEL
LIN {X 0,Y 187.456,Z 738.489,A -85,B 0,C 180,E1 -25234.435,E2 -25234.435} C_VEL
LIN {X 0,Y 192.701,Z 735.258,A -85,B 0,C 180,E1 -25235.701,E2 -25235.701} C_VEL
LIN {X 0,Y 194.452,Z 734.274,A -85,B 0,C 180,E1 -25237.336,E2 -25237.336} C_VEL
LIN {X 0,Y 192.059,Z 736.097,A -85,B 0,C 180,E1 -25238.121,E2 -25238.121} C_VEL
LIN {X 0,Y 181.239,Z 743.373,A -85,B 0,C 180,E1 -25240.877,E2 -25240.877} C_VEL
LIN {X 0,Y 170.869,Z 749.366,A -85,B 0,C 180,E1 -25243.967,E2 -25243.967} C_VEL
LIN {X 0,Y 160.835,Z 754.131,A -85,B 0,C 180,E1 -25247.37,E2 -25247.37} C_VEL
LIN {X 0,Y 154.047,Z 756.862,A -85,B 0,C 180,E1 -25250.308,E2 -25250.308} C_VEL
LIN {X 0,Y 145.874,Z 759.449,A -85,B 0,C 180,E1 -25254.683,E2 -25254.683} C_VEL
LIN {X 0,Y 139.104,Z 760.879,A -85,B 0,C 180,E1 -25259.657,E2 -25259.657} C_VEL
LIN {X 0,Y 133.79,Z 761.154,A -85,B 0,C 180,E1 -25265.154,E2 -25265.154} C_VEL
LIN {X 0,Y 129.999,Z 760.262,A -85,B 0,C 180,E1 -25271.076,E2 -25271.076} C_VEL
LIN {X 0,Y 128.052,Z 758.163,A -85,B 0,C 180,E1 -25277.321,E2 -25277.321} C_VEL
LIN {X 0,Y 127.801,Z 754.755,A -85,B 0,C 180,E1 -25283.689,E2 -25283.689} C_VEL
LIN {X 0,Y 128.331,Z 751.174,A -85,B 0,C 180,E1 -25288.434,E2 -25288.434} C_VEL
LIN {X 0,Y 128.325,Z 748.02,A -85,B 0,C 180,E1 -25291.572,E2 -25291.572} C_VEL
LIN {X 0,Y 128.289,Z 742.133,A -85,B 0,C 180,E1 -25296.293,E2 -25296.293} C_VEL
LIN {X 0,Y 128.648,Z 734.937,A -85,B 0,C 180,E1 -25300.866,E2 -25300.866} C_VEL
LIN {X 0,Y 129.453,Z 727.073,A -85,B 0,C 180,E1 -25304.947,E2 -25304.947} C_VEL
LIN {X 0,Y 130.964,Z 716.948,A -85,B 0,C 180,E1 -25309.192,E2 -25309.192} C_VEL
LIN {X 0,Y 131.635,Z 713.136,A -85,B 0,C 180,E1 -25310.717,E2 -25310.717} C_VEL
LIN {X 0,Y 132.966,Z 707.133,A -85,B 0,C 180,E1 -25314.184,E2 -25314.184} C_VEL
LIN {X 0,Y 133.902,Z 698.93,A -85,B 0,C 180,E1 -25318.191,E2 -25318.191} C_VEL
LIN {X 0,Y 135.334,Z 688.93,A -85,B 0,C 180,E1 -25322.163,E2 -25322.163} C_VEL
LIN {X 0,Y 136.791,Z 677.66,A -85,B 0,C 180,E1 -25325.765,E2 -25325.765} C_VEL
LIN {X 0,Y 137.897,Z 665.226,A -85,B 0,C 180,E1 -25329.011,E2 -25329.011} C_VEL
LIN {X 0,Y 138.404,Z 653.153,A -85,B 0,C 180,E1 -25331.555,E2 -25331.555} C_VEL
LIN {X 0,Y 137.965,Z 639.86,A -85,B 0,C 180,E1 -25333.936,E2 -25333.936} C_VEL
LIN {X 0,Y 137.261,Z 635.377,A -85,B 0,C 180,E1 -25334.758,E2 -25334.758} C_VEL
LIN {X 0,Y 135.432,Z 630.909,A -85,B 0,C 180,E1 -25335.889,E2 -25335.889} C_VEL
LIN {X 0,Y 133.629,Z 626.672,A -85,B 0,C 180,E1 -25336.948,E2 -25336.948} C_VEL
LIN {X 0,Y 133.391,Z 626.284,A -85,B 0,C 180,E1 -25337.072,E2 -25337.072} C_VEL
LIN {X 0,Y 131.327,Z 623.807,A -85,B 0,C 180,E1 -25338.123,E2 -25338.123} C_VEL
LIN {X 0,Y 127.538,Z 621.015,A -85,B 0,C 180,E1 -25340.279,E2 -25340.279} C_VEL
LIN {X 0,Y 124.554,Z 618.993,A -85,B 0,C 180,E1 -25342.898,E2 -25342.898} C_VEL
LIN {X 0,Y 123.755,Z 617.732,A -85,B 0,C 180,E1 -25344.637,E2 -25344.637} C_VEL
LIN {X 0,Y 123.149,Z 614.38,A -85,B 0,C 180,E1 -25349.093,E2 -25349.093} C_VEL
LIN {X 0,Y 122.279,Z 610.678,A -85,B 0,C 180,E1 -25354.463,E2 -25354.463} C_VEL
LIN {X 0,Y 122.03,Z 609.285,A -85,B 0,C 180,E1 -25356.857,E2 -25356.857} C_VEL
LIN {X 0,Y 122.125,Z 609.276,A -85,B 0,C 180,E1 -25363.276,E2 -25363.276} C_VEL
LIN {X 0,Y 122.372,Z 609.242,A -85,B 0,C 180,E1 -25367.522,E2 -25367.522} C_VEL
LIN {X 0,Y 122.463,Z 609.234,A -85,B 0,C 180,E1 -25370.085,E2 -25370.085} C_VEL
LIN {X 0,Y 122.615,Z 609.207,A -85,B 0,C 180,E1 -25376.713,E2 -25376.713} C_VEL
LIN {X 0,Y 123.049,Z 609.156,A -85,B 0,C 180,E1 -25379.999,E2 -25379.999} C_VEL
LIN {X 0,Y 122.421,Z 609.213,A -85,B 0,C 180,E1 -25387.184,E2 -25387.184} C_VEL
LIN {X 0,Y 122.369,Z 609.235,A -85,B 0,C 180,E1 -25392.471,E2 -25392.471} C_VEL
LIN {X 0,Y 122.051,Z 609.279,A -85,B 0,C 180,E1 -25400.211,E2 -25400.211} C_VEL
LIN {X 0,Y 121.988,Z 609.28,A -85,B 0,C 180,E1 -25403.782,E2 -25403.782} C_VEL
LIN {X 0,Y 121.943,Z 609.291,A -85,B 0,C 180,E1 -25410.169,E2 -25410.169} C_VEL
LIN {X 0,Y 121.888,Z 609.302,A -85,B 0,C 180,E1 -25416.169,E2 -25416.169} C_VEL
LIN {X 0,Y 121.883,Z 609.301,A -85,B 0,C 180,E1 -25421.44,E2 -25421.44} C_VEL
LIN {X 0,Y 121.905,Z 609.298,A -85,B 0,C 180,E1 -25428.542,E2 -25428.542} C_VEL
LIN {X 0,Y 121.959,Z 609.404,A -85,B 0,C 180,E1 -25434.053,E2 -25434.053} C_VEL
LIN {X 0,Y 122.894,Z 612.032,A -85,B 0,C 180,E1 -25435.005,E2 -25435.005} C_VEL
LIN {X 0,Y 126.36,Z 617.595,A -85,B 0,C 180,E1 -25437.687,E2 -25437.687} C_VEL
LIN {X 0,Y 130.661,Z 626.397,A -85,B 0,C 180,E1 -25441.473,E2 -25441.473} C_VEL
LIN {X 0,Y 133.708,Z 634.497,A -85,B 0,C 180,E1 -25444.781,E2 -25444.781} C_VEL
LIN {X 0,Y 136.118,Z 643.199,A -85,B 0,C 180,E1 -25448.333,E2 -25448.333} C_VEL
LIN {X 0,Y 137.426,Z 649.896,A -85,B 0,C 180,E1 -25451.145,E2 -25451.145} C_VEL
LIN {X 0,Y 136.505,Z 653.596,A -85,B 0,C 180,E1 -25452.391,E2 -25452.391} C_VEL
LIN {X 0,Y 133.66,Z 662.087,A -85,B 0,C 180,E1 -25455.534,E2 -25455.534} C_VEL
LIN {X 0,Y 130.928,Z 669.919,A -85,B 0,C 180,E1 -25459.168,E2 -25459.168} C_VEL
LIN {X 0,Y 128.042,Z 677.624,A -85,B 0,C 180,E1 -25463.695,E2 -25463.695} C_VEL
LIN {X 0,Y 125.785,Z 683.837,A -85,B 0,C 180,E1 -25468.396,E2 -25468.396} C_VEL
LIN {X 0,Y 124.132,Z 688.81,A -85,B 0,C 180,E1 -25473.243,E2 -25473.243} C_VEL
LIN {X 0,Y 123.22,Z 692.662,A -85,B 0,C 180,E1 -25478.195,E2 -25478.195} C_VEL
LIN {X 0,Y 123.06,Z 695.804,A -85,B 0,C 180,E1 -25483.867,E2 -25483.867} C_VEL
LIN {X 0,Y 123.948,Z 697.818,A -85,B 0,C 180,E1 -25489.886,E2 -25489.886} C_VEL
LIN {X 0,Y 126.232,Z 698.452,A -85,B 0,C 180,E1 -25496.446,E2 -25496.446} C_VEL
LIN {X 0,Y 127.859,Z 698.186,A -85,B 0,C 180,E1 -25499.646,E2 -25499.646} C_VEL
LIN {X 0,Y 129.829,Z 697.481,A -85,B 0,C 180,E1 -25502.77,E2 -25502.77} C_VEL
LIN {X 0,Y 134.284,Z 695.06,A -85,B 0,C 180,E1 -25508.277,E2 -25508.277} C_VEL
LIN {X 0,Y 138.816,Z 691.817,A -85,B 0,C 180,E1 -25512.698,E2 -25512.698} C_VEL
LIN {X 0,Y 139.11,Z 691.07,A -85,B 0,C 180,E1 -25513.918,E2 -25513.918} C_VEL
LIN {X 0,Y 134.329,Z 691.007,A -85,B 0,C 180,E1 -25517.146,E2 -25517.146} C_VEL
LIN {X 0,Y 130.353,Z 691.206,A -85,B 0,C 180,E1 -25519.687,E2 -25519.687} C_VEL
LIN {X 0,Y 126.993,Z 691.131,A -85,B 0,C 180,E1 -25522.502,E2 -25522.502} C_VEL
LIN {X 0,Y 125.696,Z 690.884,A -85,B 0,C 180,E1 -25524.175,E2 -25524.175} C_VEL
LIN {X 0,Y 123.529,Z 702.72,A -85,B 0,C 180,E1 -25528.345,E2 -25528.345} C_VEL
LIN {X 0,Y 121.894,Z 712.34,A -85,B 0,C 180,E1 -25532.534,E2 -25532.534} C_VEL
LIN {X 0,Y 120.584,Z 722.278,A -85,B 0,C 180,E1 -25537.92,E2 -25537.92} C_VEL
LIN {X 0,Y 119.861,Z 729.792,A -85,B 0,C 180,E1 -25542.953,E2 -25542.953} C_VEL
LIN {X 0,Y 119.66,Z 736.033,A -85,B 0,C 180,E1 -25548.139,E2 -25548.139} C_VEL
LIN {X 0,Y 120.234,Z 741.345,A -85,B 0,C 180,E1 -25553.533,E2 -25553.533} C_VEL
LIN {X 0,Y 122.098,Z 746.373,A -85,B 0,C 180,E1 -25560.001,E2 -25560.001} C_VEL
LIN {X 0,Y 125.594,Z 750.132,A -85,B 0,C 180,E1 -25566.427,E2 -25566.427} C_VEL
LIN {X 0,Y 130.672,Z 752.571,A -85,B 0,C 180,E1 -25572.425,E2 -25572.425} C_VEL
LIN {X 0,Y 137.245,Z 753.67,A -85,B 0,C 180,E1 -25577.895,E2 -25577.895} C_VEL
LIN {X 0,Y 145.187,Z 753.472,A -85,B 0,C 180,E1 -25582.785,E2 -25582.785} C_VEL
LIN {X 0,Y 154.314,Z 751.975,A -85,B 0,C 180,E1 -25587.094,E2 -25587.094} C_VEL
LIN {X 0,Y 164.411,Z 749.158,A -85,B 0,C 180,E1 -25590.862,E2 -25590.862} C_VEL
LIN {X 0,Y 175.436,Z 744.824,A -85,B 0,C 180,E1 -25594.115,E2 -25594.115} C_VEL
LIN {X 0,Y 186.218,Z 739.465,A -85,B 0,C 180,E1 -25596.724,E2 -25596.724} C_VEL
LIN {X 0,Y 185.163,Z 740.13,A -85,B 0,C 180,E1 -25597.153,E2 -25597.153} C_VEL
LIN {X 0,Y 174.061,Z 746.548,A -85,B 0,C 180,E1 -25599.905,E2 -25599.905} C_VEL
LIN {X 0,Y 163.41,Z 751.725,A -85,B 0,C 180,E1 -25603.022,E2 -25603.022} C_VEL
LIN {X 0,Y 153.263,Z 755.704,A -85,B 0,C 180,E1 -25606.545,E2 -25606.545} C_VEL
LIN {X 0,Y 144.301,Z 758.468,A -85,B 0,C 180,E1 -25610.721,E2 -25610.721} C_VEL
LIN {X 0,Y 136.366,Z 760.077,A -85,B 0,C 180,E1 -25615.468,E2 -25615.468} C_VEL
LIN {X 0,Y 129.992,Z 760.567,A -85,B 0,C 180,E1 -25620.887,E2 -25620.887} C_VEL
LIN {X 0,Y 125.092,Z 759.913,A -85,B 0,C 180,E1 -25626.845,E2 -25626.845} C_VEL
LIN {X 0,Y 122.077,Z 758.14,A -85,B 0,C 180,E1 -25633.274,E2 -25633.274} C_VEL
LIN {X 0,Y 120.873,Z 755.12,A -85,B 0,C 180,E1 -25639.958,E2 -25639.958} C_VEL
LIN {X 0,Y 121.034,Z 751.959,A -85,B 0,C 180,E1 -25645.006,E2 -25645.006} C_VEL
LIN {X 0,Y 121.473,Z 749.302,A -85,B 0,C 180,E1 -25648.345,E2 -25648.345} C_VEL
LIN {X 0,Y 121.414,Z 745.966,A -85,B 0,C 180,E1 -25651.662,E2 -25651.662} C_VEL
LIN {X 0,Y 121.389,Z 739.721,A -85,B 0,C 180,E1 -25656.652,E2 -25656.652} C_VEL
LIN {X 0,Y 121.745,Z 732.896,A -85,B 0,C 180,E1 -25661.074,E2 -25661.074} C_VEL
LIN {X 0,Y 122.768,Z 723.922,A -85,B 0,C 180,E1 -25665.782,E2 -25665.782} C_VEL
LIN {X 0,Y 124.193,Z 714.542,A -85,B 0,C 180,E1 -25669.852,E2 -25669.852} C_VEL
LIN {X 0,Y 125.754,Z 708.361,A -85,B 0,C 180,E1 -25673.905,E2 -25673.905} C_VEL
LIN {X 0,Y 126.837,Z 700.1,A -85,B 0,C 180,E1 -25678.371,E2 -25678.371} C_VEL
LIN {X 0,Y 128.425,Z 690.159,A -85,B 0,C 180,E1 -25682.714,E2 -25682.714} C_VEL
LIN {X 0,Y 130.044,Z 679.502,A -85,B 0,C 180,E1 -25686.478,E2 -25686.478} C_VEL
LIN {X 0,Y 131.244,Z 669.145,A -85,B 0,C 180,E1 -25689.49,E2 -25689.49} C_VEL
LIN {X 0,Y 132.126,Z 657.325,A -85,B 0,C 180,E1 -25692.327,E2 -25692.327} C_VEL
LIN {X 0,Y 132.234,Z 644.097,A -85,B 0,C 180,E1 -25694.996,E2 -25694.996} C_VEL
LIN {X 0,Y 131.706,Z 638.611,A -85,B 0,C 180,E1 -25696.075,E2 -25696.075} C_VEL
LIN {X 0,Y 128.402,Z 630.308,A -85,B 0,C 180,E1 -25698.437,E2 -25698.437} C_VEL
LIN {X 0,Y 126.311,Z 625.467,A -85,B 0,C 180,E1 -25699.827,E2 -25699.827} C_VEL
LIN {X 0,Y 124.524,Z 621.647,A -85,B 0,C 180,E1 -25700.974,E2 -25700.974} C_VEL
LIN {X 0,Y 124.22,Z 620.414,A -85,B 0,C 180,E1 -25701.251,E2 -25701.251} C_VEL
LIN {X 0,Y 123.755,Z 617.732,A -85,B 0,C 180,E1 -25704.637,E2 -25704.637} C_VEL
LIN {X 0,Y 122.836,Z 616.595,A -85,B 0,C 180,E1 -25706.335,E2 -25706.335} C_VEL
LIN {X 0,Y 119.658,Z 615.283,A -85,B 0,C 180,E1 -25709.045,E2 -25709.045} C_VEL
LIN {X 0,Y 116.437,Z 613.999,A -85,B 0,C 180,E1 -25711.9,E2 -25711.9} C_VEL
LIN {X 0,Y 115.519,Z 612.946,A -85,B 0,C 180,E1 -25713.773,E2 -25713.773} C_VEL
LIN {X 0,Y 115.003,Z 610.161,A -85,B 0,C 180,E1 -25718.488,E2 -25718.488} C_VEL
LIN {X 0,Y 115.155,Z 610.146,A -85,B 0,C 180,E1 -25725.869,E2 -25725.869} C_VEL
LIN {X 0,Y 115.4,Z 610.114,A -85,B 0,C 180,E1 -25729.471,E2 -25729.471} C_VEL
LIN {X 0,Y 115.541,Z 610.088,A -85,B 0,C 180,E1 -25736.511,E2 -25736.511} C_VEL
LIN {X 0,Y 116.001,Z 610.034,A -85,B 0,C 180,E1 -25739.999,E2 -25739.999} C_VEL
LIN {X 0,Y 115.387,Z 610.091,A -85,B 0,C 180,E1 -25747.087,E2 -25747.087} C_VEL
LIN {X 0,Y 115.29,Z 610.114,A -85,B 0,C 180,E1 -25752.736,E2 -25752.736} C_VEL
LIN {X 0,Y 115.018,Z 610.134,A -85,B 0,C 180,E1 -25757.788,E2 -25757.788} C_VEL
LIN {X 0,Y 114.952,Z 610.158,A -85,B 0,C 180,E1 -25763.49,E2 -25763.49} C_VEL
LIN {X 0,Y 114.866,Z 610.177,A -85,B 0,C 180,E1 -25771.06,E2 -25771.06} C_VEL
LIN {X 0,Y 114.785,Z 610.183,A -85,B 0,C 180,E1 -25777.752,E2 -25777.752} C_VEL
LIN {X 0,Y 114.796,Z 610.174,A -85,B 0,C 180,E1 -25782.717,E2 -25782.717} C_VEL
LIN {X 0,Y 114.847,Z 610.172,A -85,B 0,C 180,E1 -25789.961,E2 -25789.961} C_VEL
LIN {X 0,Y 114.869,Z 610.231,A -85,B 0,C 180,E1 -25790.435,E2 -25790.435} C_VEL
LIN {X 0,Y 115.785,Z 612.961,A -85,B 0,C 180,E1 -25791.538,E2 -25791.538} C_VEL
LIN {X 0,Y 117.156,Z 614.584,A -85,B 0,C 180,E1 -25792.638,E2 -25792.638} C_VEL
LIN {X 0,Y 121.836,Z 623.057,A -85,B 0,C 180,E1 -25796.996,E2 -25796.996} C_VEL
LIN {X 0,Y 125.219,Z 630.332,A -85,B 0,C 180,E1 -25800.447,E2 -25800.447} C_VEL
LIN {X 0,Y 128.272,Z 639.239,A -85,B 0,C 180,E1 -25804.413,E2 -25804.413} C_VEL
LIN {X 0,Y 130.137,Z 646.828,A -85,B 0,C 180,E1 -25807.785,E2 -25807.785} C_VEL
LIN {X 0,Y 130.962,Z 651.851,A -85,B 0,C 180,E1 -25810.074,E2 -25810.074} C_VEL
LIN {X 0,Y 128.133,Z 660.558,A -85,B 0,C 180,E1 -25813.261,E2 -25813.261} C_VEL
LIN {X 0,Y 125.06,Z 668.821,A -85,B 0,C 180,E1 -25817.007,E2 -25817.007} C_VEL
LIN {X 0,Y 121.949,Z 676.933,A -85,B 0,C 180,E1 -25821.713,E2 -25821.713} C_VEL
LIN {X 0,Y 119.375,Z 683.514,A -85,B 0,C 180,E1 -25826.622,E2 -25826.622} C_VEL
LIN {X 0,Y 117.471,Z 688.773,A -85,B 0,C 180,E1 -25831.711,E2 -25831.711} C_VEL
LIN {X 0,Y 116.331,Z 692.883,A -85,B 0,C 180,E1 -25836.937,E2 -25836.937} C_VEL
LIN {X 0,Y 115.999,Z 695.019,A -85,B 0,C 180,E1 -25840.469,E2 -25840.469} C_VEL
LIN {X 0,Y 116.054,Z 696.874,A -85,B 0,C 180,E1 -25844.326,E2 -25844.326} C_VEL
LIN {X 0,Y 116.423,Z 698.056,A -85,B 0,C 180,E1 -25847.564,E2 -25847.564} C_VEL
LIN {X 0,Y 117.186,Z 698.923,A -85,B 0,C 180,E1 -25851.087,E2 -25851.087} C_VEL
LIN {X 0,Y 119.767,Z 699.471,A -85,B 0,C 180,E1 -25857.994,E2 -25857.994} C_VEL
LIN {X 0,Y 121.603,Z 699.14,A -85,B 0,C 180,E1 -25861.339,E2 -25861.339} C_VEL
LIN {X 0,Y 123.773,Z 698.36,A -85,B 0,C 180,E1 -25864.594,E2 -25864.594} C_VEL
LIN {X 0,Y 128.271,Z 696.059,A -85,B 0,C 180,E1 -25869.911,E2 -25869.911} C_VEL
LIN {X 0,Y 130.664,Z 694.556,A -85,B 0,C 180,E1 -25872.243,E2 -25872.243} C_VEL
LIN {X 0,Y 131.427,Z 693.674,A -85,B 0,C 180,E1 -25873.792,E2 -25873.792} C_VEL
LIN {X 0,Y 121.846,Z 694.069,A -85,B 0,C 180,E1 -25880.621,E2 -25880.621} C_VEL
LIN {X 0,Y 118.183,Z 693.956,A -85,B 0,C 180,E1 -25884.565,E2 -25884.565} C_VEL
LIN {X 0,Y 118.018,Z 693.916,A -85,B 0,C 180,E1 -25885.16,E2 -25885.16} C_VEL
LIN {X 0,Y 116.042,Z 704.167,A -85,B 0,C 180,E1 -25889.11,E2 -25889.11} C_VEL
LIN {X 0,Y 114.319,Z 715.341,A -85,B 0,C 180,E1 -25894.512,E2 -25894.512} C_VEL
LIN {X 0,Y 113.394,Z 722.709,A -85,B 0,C 180,E1 -25898.907,E2 -25898.907} C_VEL
LIN {X 0,Y 112.726,Z 730.57,A -85,B 0,C 180,E1 -25904.636,E2 -25904.636} C_VEL
LIN {X 0,Y 112.834,Z 737.608,A -85,B 0,C 180,E1 -25911.043,E2 -25911.043} C_VEL
LIN {X 0,Y 113.842,Z 742.454,A -85,B 0,C 180,E1 -25916.462,E2 -25916.462} C_VEL
LIN {X 0,Y 116.483,Z 747.444,A -85,B 0,C 180,E1 -25923.46,E2 -25923.46} C_VEL
LIN {X 0,Y 120.818,Z 751.045,A -85,B 0,C 180,E1 -25930.051,E2 -25930.051} C_VEL
LIN {X 0,Y 126.799,Z 753.315,A -85,B 0,C 180,E1 -25936.09,E2 -25936.09} C_VEL
LIN {X 0,Y 134.316,Z 754.3,A -85,B 0,C 180,E1 -25941.487,E2 -25941.487} C_VEL
LIN {X 0,Y 143.074,Z 754.019,A -85,B 0,C 180,E1 -25946.239,E2 -25946.239} C_VEL
LIN {X 0,Y 153.021,Z 752.466,A -85,B 0,C 180,E1 -25950.347,E2 -25950.347} C_VEL
LIN {X 0,Y 163.85,Z 749.532,A -85,B 0,C 180,E1 -25953.892,E2 -25953.892} C_VEL
LIN {X 0,Y 173.571,Z 745.967,A -85,B 0,C 180,E1 -25956.456,E2 -25956.456} C_VEL
LIN {X 0,Y 171.895,Z 746.919,A -85,B 0,C 180,E1 -25957.531,E2 -25957.531} C_VEL
LIN {X 0,Y 161.441,Z 751.589,A -85,B 0,C 180,E1 -25960.379,E2 -25960.379} C_VEL
LIN {X 0,Y 153.336,Z 754.532,A -85,B 0,C 180,E1 -25962.836,E2 -25962.836} C_VEL
LIN {X 0,Y 143.421,Z 757.457,A -85,B 0,C 180,E1 -25966.687,E2 -25966.687} C_VEL
LIN {X 0,Y 134.556,Z 759.26,A -85,B 0,C 180,E1 -25971.191,E2 -25971.191} C_VEL
LIN {X 0,Y 127.053,Z 759.953,A -85,B 0,C 180,E1 -25976.42,E2 -25976.42} C_VEL
LIN {X 0,Y 121.095,Z 759.542,A -85,B 0,C 180,E1 -25982.339,E2 -25982.339} C_VEL
LIN {X 0,Y 116.76,Z 757.996,A -85,B 0,C 180,E1 -25988.833,E2 -25988.833} C_VEL
LIN {X 0,Y 114.461,Z 755.312,A -85,B 0,C 180,E1 -25995.786,E2 -25995.786} C_VEL
LIN {X 0,Y 114.087,Z 751.329,A -85,B 0,C 180,E1 -26002.926,E2 -26002.926} C_VEL
LIN {X 0,Y 114.626,Z 747.307,A -85,B 0,C 180,E1 -26008.247,E2 -26008.247} C_VEL
LIN {X 0,Y 114.512,Z 742.801,A -85,B 0,C 180,E1 -26012.641,E2 -26012.641} C_VEL
LIN {X 0,Y 114.572,Z 735.903,A -85,B 0,C 180,E1 -26017.936,E2 -26017.936} C_VEL
LIN {X 0,Y 115.193,Z 727.551,A -85,B 0,C 180,E1 -26023.089,E2 -26023.089} C_VEL
LIN {X 0,Y 116.344,Z 718.602,A -85,B 0,C 180,E1 -26027.583,E2 -26027.583} C_VEL
LIN {X 0,Y 116.788,Z 715.742,A -85,B 0,C 180,E1 -26028.875,E2 -26028.875} C_VEL
LIN {X 0,Y 118.766,Z 708.083,A -85,B 0,C 180,E1 -26034.474,E2 -26034.474} C_VEL
LIN {X 0,Y 119.836,Z 700.661,A -85,B 0,C 180,E1 -26038.843,E2 -26038.843} C_VEL
LIN {X 0,Y 121.522,Z 691.3,A -85,B 0,C 180,E1 -26043.33,E2 -26043.33} C_VEL
LIN {X 0,Y 123.427,Z 680.252,A -85,B 0,C 180,E1 -26047.568,E2 -26047.568} C_VEL
LIN {X 0,Y 125.057,Z 668.172,A -85,B 0,C 180,E1 -26051.329,E2 -26051.329} C_VEL
LIN {X 0,Y 126.061,Z 657.341,A -85,B 0,C 180,E1 -26054.083,E2 -26054.083} C_VEL
LIN {X 0,Y 126.357,Z 644.107,A -85,B 0,C 180,E1 -26056.941,E2 -26056.941} C_VEL
LIN {X 0,Y 126.176,Z 641.768,A -85,B 0,C 180,E1 -26057.462,E2 -26057.462} C_VEL
LIN {X 0,Y 123.216,Z 633.951,A -85,B 0,C 180,E1 -26059.948,E2 -26059.948} C_VEL
LIN {X 0,Y 121.433,Z 629.495,A -85,B 0,C 180,E1 -26061.39,E2 -26061.39} C_VEL
LIN {X 0,Y 119.293,Z 624.543,A -85,B 0,C 180,E1 -26063.041,E2 -26063.041} C_VEL
LIN {X 0,Y 117.282,Z 620.718,A -85,B 0,C 180,E1 -26064.512,E2 -26064.512} C_VEL
LIN {X 0,Y 116.753,Z 618.87,A -85,B 0,C 180,E1 -26065.119,E2 -26065.119} C_VEL
LIN {X 0,Y 115.892,Z 614.778,A -85,B 0,C 180,E1 -26070.977,E2 -26070.977} C_VEL
LIN {X 0,Y 115.519,Z 612.946,A -85,B 0,C 180,E1 -26073.773,E2 -26073.773} C_VEL
LIN {X 0,Y 114.591,Z 611.601,A -85,B 0,C 180,E1 -26076.582,E2 -26076.582} C_VEL
LIN {X 0,Y 112.95,Z 610.945,A -85,B 0,C 180,E1 -26079.428,E2 -26079.428} C_VEL
LIN {X 0,Y 108.609,Z 610.956,A -85,B 0,C 180,E1 -26087.452,E2 -26087.452} C_VEL
LIN {X 0,Y 108.281,Z 610.993,A -85,B 0,C 180,E1 -26089.578,E2 -26089.578} C_VEL
LIN {X 0,Y 108.467,Z 610.969,A -85,B 0,C 180,E1 -26096.284,E2 -26096.284} C_VEL
LIN {X 0,Y 108.951,Z 610.912,A -85,B 0,C 180,E1 -26099.999,E2 -26099.999} C_VEL
LIN {X 0,Y 108.337,Z 610.972,A -85,B 0,C 180,E1 -26107.453,E2 -26107.453} C_VEL
LIN {X 0,Y 108.207,Z 610.992,A -85,B 0,C 180,E1 -26113.018,E2 -26113.018} C_VEL
LIN {X 0,Y 107.91,Z 611.03,A -85,B 0,C 180,E1 -26119.003,E2 -26119.003} C_VEL
LIN {X 0,Y 107.864,Z 611.034,A -85,B 0,C 180,E1 -26124.183,E2 -26124.183} C_VEL
LIN {X 0,Y 107.788,Z 611.059,A -85,B 0,C 180,E1 -26132.04,E2 -26132.04} C_VEL
LIN {X 0,Y 107.694,Z 611.064,A -85,B 0,C 180,E1 -26138.449,E2 -26138.449} C_VEL
LIN {X 0,Y 107.708,Z 611.174,A -85,B 0,C 180,E1 -26145.964,E2 -26145.964} C_VEL
LIN {X 0,Y 108.678,Z 613.728,A -85,B 0,C 180,E1 -26147.261,E2 -26147.261} C_VEL
LIN {X 0,Y 110.861,Z 616.422,A -85,B 0,C 180,E1 -26149.378,E2 -26149.378} C_VEL
LIN {X 0,Y 111.789,Z 618.458,A -85,B 0,C 180,E1 -26150.496,E2 -26150.496} C_VEL
LIN {X 0,Y 114.294,Z 622.563,A -85,B 0,C 180,E1 -26153.068,E2 -26153.068} C_VEL
LIN {X 0,Y 118.469,Z 631.036,A -85,B 0,C 180,E1 -26157.726,E2 -26157.726} C_VEL
LIN {X 0,Y 121.388,Z 639.131,A -85,B 0,C 180,E1 -26161.755,E2 -26161.755} C_VEL
LIN {X 0,Y 123.456,Z 647.08,A -85,B 0,C 180,E1 -26165.617,E2 -26165.617} C_VEL
LIN {X 0,Y 124.547,Z 653.794,A -85,B 0,C 180,E1 -26168.901,E2 -26168.901} C_VEL
LIN {X 0,Y 121.408,Z 662.577,A -85,B 0,C 180,E1 -26172.304,E2 -26172.304} C_VEL
LIN {X 0,Y 118.209,Z 670.673,A -85,B 0,C 180,E1 -26176.239,E2 -26176.239} C_VEL
LIN {X 0,Y 114.922,Z 678.656,A -85,B 0,C 180,E1 -26181.203,E2 -26181.203} C_VEL
LIN {X 0,Y 112.269,Z 685.073,A -85,B 0,C 180,E1 -26186.408,E2 -26186.408} C_VEL
LIN {X 0,Y 110.337,Z 690.207,A -85,B 0,C 180,E1 -26191.822,E2 -26191.822} C_VEL
LIN {X 0,Y 109.211,Z 694.218,A -85,B 0,C 180,E1 -26197.391,E2 -26197.391} C_VEL
LIN {X 0,Y 108.93,Z 696.307,A -85,B 0,C 180,E1 -26201.157,E2 -26201.157} C_VEL
LIN {X 0,Y 109.054,Z 697.979,A -85,B 0,C 180,E1 -26204.935,E2 -26204.935} C_VEL
LIN {X 0,Y 109.577,Z 699.216,A -85,B 0,C 180,E1 -26208.701,E2 -26208.701} C_VEL
LIN {X 0,Y 111.72,Z 700.458,A -85,B 0,C 180,E1 -26216.122,E2 -26216.122} C_VEL
LIN {X 0,Y 113.494,Z 700.479,A -85,B 0,C 180,E1 -26219.898,E2 -26219.898} C_VEL
LIN {X 0,Y 117.847,Z 699.246,A -85,B 0,C 180,E1 -26226.606,E2 -26226.606} C_VEL
LIN {X 0,Y 122.421,Z 697.047,A -85,B 0,C 180,E1 -26231.731,E2 -26231.731} C_VEL
LIN {X 0,Y 123.709,Z 696.322,A -85,B 0,C 180,E1 -26232.974,E2 -26232.974} C_VEL
LIN {X 0,Y 120.53,Z 696.382,A -85,B 0,C 180,E1 -26235.598,E2 -26235.598} C_VEL
LIN {X 0,Y 113.406,Z 696.751,A -85,B 0,C 180,E1 -26241.706,E2 -26241.706} C_VEL
LIN {X 0,Y 110.409,Z 696.62,A -85,B 0,C 180,E1 -26245.836,E2 -26245.836} C_VEL
LIN {X 0,Y 110.309,Z 696.748,A -85,B 0,C 180,E1 -26246.218,E2 -26246.218} C_VEL
LIN {X 0,Y 108.31,Z 707.386,A -85,B 0,C 180,E1 -26250.88,E2 -26250.88} C_VEL
LIN {X 0,Y 107.003,Z 716.403,A -85,B 0,C 180,E1 -26255.765,E2 -26255.765} C_VEL
LIN {X 0,Y 106.054,Z 725.246,A -85,B 0,C 180,E1 -26261.654,E2 -26261.654} C_VEL
LIN {X 0,Y 105.683,Z 732.389,A -85,B 0,C 180,E1 -26267.52,E2 -26267.52} C_VEL
LIN {X 0,Y 106.289,Z 738.973,A -85,B 0,C 180,E1 -26274.238,E2 -26274.238} C_VEL
LIN {X 0,Y 107.79,Z 743.655,A -85,B 0,C 180,E1 -26280.001,E2 -26280.001} C_VEL
LIN {X 0,Y 111.299,Z 748.454,A -85,B 0,C 180,E1 -26287.257,E2 -26287.257} C_VEL
LIN {X 0,Y 116.607,Z 751.897,A -85,B 0,C 180,E1 -26293.952,E2 -26293.952} C_VEL
LIN {X 0,Y 123.52,Z 754.031,A -85,B 0,C 180,E1 -26299.963,E2 -26299.963} C_VEL
LIN {X 0,Y 132.209,Z 754.945,A -85,B 0,C 180,E1 -26305.36,E2 -26305.36} C_VEL
LIN {X 0,Y 141.591,Z 754.594,A -85,B 0,C 180,E1 -26309.761,E2 -26309.761} C_VEL
LIN {X 0,Y 152.251,Z 752.971,A -85,B 0,C 180,E1 -26313.638,E2 -26313.638} C_VEL
LIN {X 0,Y 161.86,Z 750.578,A -85,B 0,C 180,E1 -26316.418,E2 -26316.418} C_VEL
LIN {X 0,Y 161.12,Z 750.975,A -85,B 0,C 180,E1 -26317.319,E2 -26317.319} C_VEL
LIN {X 0,Y 148.625,Z 755.082,A -85,B 0,C 180,E1 -26320.84,E2 -26320.84} C_VEL
LIN {X 0,Y 138.354,Z 757.565,A -85,B 0,C 180,E1 -26324.675,E2 -26324.675} C_VEL
LIN {X 0,Y 129.11,Z 758.957,A -85,B 0,C 180,E1 -26329.22,E2 -26329.22} C_VEL
LIN {X 0,Y 121.222,Z 759.275,A -85,B 0,C 180,E1 -26334.57,E2 -26334.57} C_VEL
LIN {X 0,Y 114.889,Z 758.532,A -85,B 0,C 180,E1 -26340.704,E2 -26340.704} C_VEL
LIN {X 0,Y 110.254,Z 756.69,A -85,B 0,C 180,E1 -26347.517,E2 -26347.517} C_VEL
LIN {X 0,Y 107.749,Z 753.713,A -85,B 0,C 180,E1 -26354.88,E2 -26354.88} C_VEL
LIN {X 0,Y 107.276,Z 749.47,A -85,B 0,C 180,E1 -26362.475,E2 -26362.475} C_VEL
LIN {X 0,Y 107.804,Z 745.168,A -85,B 0,C 180,E1 -26368.136,E2 -26368.136} C_VEL
LIN {X 0,Y 107.684,Z 739.296,A -85,B 0,C 180,E1 -26373.745,E2 -26373.745} C_VEL
LIN {X 0,Y 107.778,Z 731.978,A -85,B 0,C 180,E1 -26379.238,E2 -26379.238} C_VEL
LIN {X 0,Y 108.702,Z 722.333,A -85,B 0,C 180,E1 -26384.991,E2 -26384.991} C_VEL
LIN {X 0,Y 109.445,Z 716.805,A -85,B 0,C 180,E1 -26387.763,E2 -26387.763} C_VEL
LIN {X 0,Y 111.012,Z 710.288,A -85,B 0,C 180,E1 -26393.312,E2 -26393.312} C_VEL
LIN {X 0,Y 111.972,Z 706.414,A -85,B 0,C 180,E1 -26396.066,E2 -26396.066} C_VEL
LIN {X 0,Y 113.659,Z 696.925,A -85,B 0,C 180,E1 -26401.712,E2 -26401.712} C_VEL
LIN {X 0,Y 115.633,Z 687.148,A -85,B 0,C 180,E1 -26406.345,E2 -26406.345} C_VEL
LIN {X 0,Y 117.581,Z 677.01,A -85,B 0,C 180,E1 -26410.22,E2 -26410.22} C_VEL
LIN {X 0,Y 119.247,Z 665.479,A -85,B 0,C 180,E1 -26413.833,E2 -26413.833} C_VEL
LIN {X 0,Y 120.289,Z 654.156,A -85,B 0,C 180,E1 -26416.796,E2 -26416.796} C_VEL
LIN {X 0,Y 120.631,Z 646.069,A -85,B 0,C 180,E1 -26418.659,E2 -26418.659} C_VEL
LIN {X 0,Y 120.466,Z 644.373,A -85,B 0,C 180,E1 -26419.09,E2 -26419.09} C_VEL
LIN {X 0,Y 116.298,Z 632.878,A -85,B 0,C 180,E1 -26423.225,E2 -26423.225} C_VEL
LIN {X 0,Y 114.734,Z 628.995,A -85,B 0,C 180,E1 -26424.682,E2 -26424.682} C_VEL
LIN {X 0,Y 112.663,Z 624.227,A -85,B 0,C 180,E1 -26426.572,E2 -26426.572} C_VEL
LIN {X 0,Y 109.988,Z 619.606,A -85,B 0,C 180,E1 -26428.847,E2 -26428.847} C_VEL
LIN {X 0,Y 109.194,Z 617.19,A -85,B 0,C 180,E1 -26429.811,E2 -26429.811} C_VEL
LIN {X 0,Y 108.499,Z 613.973,A -85,B 0,C 180,E1 -26435.081,E2 -26435.081} C_VEL
LIN {X 0,Y 107.917,Z 611.044,A -85,B 0,C 180,E1 -26440.501,E2 -26440.501} C_VEL
LIN {X 0,Y 108.313,Z 610.994,A -85,B 0,C 180,E1 -26448.774,E2 -26448.774} C_VEL
LIN {X 0,Y 108.281,Z 610.993,A -85,B 0,C 180,E1 -26449.578,E2 -26449.578} C_VEL
LIN {X 0,Y 107.568,Z 611.085,A -85,B 0,C 180,E1 -26452.694,E2 -26452.694} C_VEL
LIN {X 0,Y 106.003,Z 611.283,A -85,B 0,C 180,E1 -26455.78,E2 -26455.78} C_VEL
LIN {X 0,Y 101.568,Z 611.802,A -85,B 0,C 180,E1 -26464.378,E2 -26464.378} C_VEL
LIN {X 0,Y 101.258,Z 611.845,A -85,B 0,C 180,E1 -26466.66,E2 -26466.66} C_VEL
LIN {X 0,Y 101.133,Z 611.868,A -85,B 0,C 180,E1 -26473.356,E2 -26473.356} C_VEL
LIN {X 0,Y 100.821,Z 611.923,A -85,B 0,C 180,E1 -26480.396,E2 -26480.396} C_VEL
LIN {X 0,Y 100.779,Z 611.908,A -85,B 0,C 180,E1 -26484.956,E2 -26484.956} C_VEL
LIN {X 0,Y 100.695,Z 611.938,A -85,B 0,C 180,E1 -26493.113,E2 -26493.113} C_VEL
LIN {X 0,Y 100.655,Z 612.067,A -85,B 0,C 180,E1 -26500.332,E2 -26500.332} C_VEL
LIN {X 0,Y 101.596,Z 614.761,A -85,B 0,C 180,E1 -26501.944,E2 -26501.944} C_VEL
LIN {X 0,Y 104.053,Z 617.389,A -85,B 0,C 180,E1 -26504.785,E2 -26504.785} C_VEL
LIN {X 0,Y 105.71,Z 620.475,A -85,B 0,C 180,E1 -26506.995,E2 -26506.995} C_VEL
LIN {X 0,Y 106.677,Z 621.565,A -85,B 0,C 180,E1 -26508.024,E2 -26508.024} C_VEL
LIN {X 0,Y 110.511,Z 629.057,A -85,B 0,C 180,E1 -26512.929,E2 -26512.929} C_VEL
LIN {X 0,Y 113.872,Z 636.894,A -85,B 0,C 180,E1 -26517.547,E2 -26517.547} C_VEL
LIN {X 0,Y 116.165,Z 644.548,A -85,B 0,C 180,E1 -26521.665,E2 -26521.665} C_VEL
LIN {X 0,Y 117.848,Z 652.789,A -85,B 0,C 180,E1 -26526.045,E2 -26526.045} C_VEL
LIN {X 0,Y 118.153,Z 655.729,A -85,B 0,C 180,E1 -26527.607,E2 -26527.607} C_VEL
LIN {X 0,Y 114.682,Z 664.564,A -85,B 0,C 180,E1 -26531.229,E2 -26531.229} C_VEL
LIN {X 0,Y 111.359,Z 672.494,A -85,B 0,C 180,E1 -26535.374,E2 -26535.374} C_VEL
LIN {X 0,Y 107.884,Z 680.309,A -85,B 0,C 180,E1 -26540.624,E2 -26540.624} C_VEL
LIN {X 0,Y 105.158,Z 686.589,A -85,B 0,C 180,E1 -26546.164,E2 -26546.164} C_VEL
LIN {X 0,Y 103.179,Z 691.625,A -85,B 0,C 180,E1 -26551.948,E2 -26551.948} C_VEL
LIN {X 0,Y 102.089,Z 695.542,A -85,B 0,C 180,E1 -26557.91,E2 -26557.91} C_VEL
LIN {X 0,Y 102.041,Z 698.981,A -85,B 0,C 180,E1 -26565.375,E2 -26565.375} C_VEL
LIN {X 0,Y 102.773,Z 700.36,A -85,B 0,C 180,E1 -26569.99,E2 -26569.99} C_VEL
LIN {X 0,Y 105.256,Z 701.521,A -85,B 0,C 180,E1 -26577.861,E2 -26577.861} C_VEL
LIN {X 0,Y 107.174,Z 701.471,A -85,B 0,C 180,E1 -26581.637,E2 -26581.637} C_VEL
LIN {X 0,Y 112.094,Z 700.132,A -85,B 0,C 180,E1 -26588.822,E2 -26588.822} C_VEL
LIN {X 0,Y 115.118,Z 698.847,A -85,B 0,C 180,E1 -26592.182,E2 -26592.182} C_VEL
LIN {X 0,Y 115.603,Z 698.474,A -85,B 0,C 180,E1 -26593.155,E2 -26593.155} C_VEL
LIN {X 0,Y 108.122,Z 699.09,A -85,B 0,C 180,E1 -26599.46,E2 -26599.46} C_VEL
LIN {X 0,Y 102.75,Z 699.211,A -85,B 0,C 180,E1 -26606.827,E2 -26606.827} C_VEL
LIN {X 0,Y 102.591,Z 699.353,A -85,B 0,C 180,E1 -26607.499,E2 -26607.499} C_VEL
LIN {X 0,Y 100.684,Z 710.442,A -85,B 0,C 180,E1 -26613.019,E2 -26613.019} C_VEL
LIN {X 0,Y 99.415,Z 720.484,A -85,B 0,C 180,E1 -26619.302,E2 -26619.302} C_VEL
LIN {X 0,Y 98.854,Z 727.251,A -85,B 0,C 180,E1 -26624.539,E2 -26624.539} C_VEL
LIN {X 0,Y 98.962,Z 734.998,A -85,B 0,C 180,E1 -26631.836,E2 -26631.836} C_VEL
LIN {X 0,Y 100.096,Z 740.409,A -85,B 0,C 180,E1 -26637.99,E2 -26637.99} C_VEL
LIN {X 0,Y 103.129,Z 746.046,A -85,B 0,C 180,E1 -26645.869,E2 -26645.869} C_VEL
LIN {X 0,Y 108.452,Z 750.559,A -85,B 0,C 180,E1 -26653.598,E2 -26653.598} C_VEL
LIN {X 0,Y 112.983,Z 752.679,A -85,B 0,C 180,E1 -26658.122,E2 -26658.122} C_VEL
LIN {X 0,Y 120.905,Z 754.74,A -85,B 0,C 180,E1 -26664.011,E2 -26664.011} C_VEL
LIN {X 0,Y 130.211,Z 755.579,A -85,B 0,C 180,E1 -26669.064,E2 -26669.064} C_VEL
LIN {X 0,Y 140.723,Z 755.179,A -85,B 0,C 180,E1 -26673.325,E2 -26673.325} C_VEL
LIN {X 0,Y 146.278,Z 754.51,A -85,B 0,C 180,E1 -26675.209,E2 -26675.209} C_VEL
LIN {X 0,Y 149.767,Z 754.061,A -85,B 0,C 180,E1 -26677.089,E2 -26677.089} C_VEL
LIN {X 0,Y 138.612,Z 756.664,A -85,B 0,C 180,E1 -26680.493,E2 -26680.493} C_VEL
LIN {X 0,Y 128.547,Z 758.182,A -85,B 0,C 180,E1 -26684.709,E2 -26684.709} C_VEL
LIN {X 0,Y 119.468,Z 758.644,A -85,B 0,C 180,E1 -26689.681,E2 -26689.681} C_VEL
LIN {X 0,Y 111.949,Z 758.075,A -85,B 0,C 180,E1 -26695.602,E2 -26695.602} C_VEL
LIN {X 0,Y 106.048,Z 756.457,A -85,B 0,C 180,E1 -26702.365,E2 -26702.365} C_VEL
LIN {X 0,Y 102.232,Z 753.757,A -85,B 0,C 180,E1 -26709.9,E2 -26709.9} C_VEL
LIN {X 0,Y 100.538,Z 749.719,A -85,B 0,C 180,E1 -26718.148,E2 -26718.148} C_VEL
LIN {X 0,Y 100.906,Z 744.598,A -85,B 0,C 180,E1 -26726.01,E2 -26726.01} C_VEL
LIN {X 0,Y 100.95,Z 740.97,A -85,B 0,C 180,E1 -26730.004,E2 -26730.004} C_VEL
LIN {X 0,Y 100.816,Z 735.41,A -85,B 0,C 180,E1 -26735.003,E2 -26735.003} C_VEL
LIN {X 0,Y 101.125,Z 727.115,A -85,B 0,C 180,E1 -26741.022,E2 -26741.022} C_VEL
LIN {X 0,Y 102.202,Z 717.471,A -85,B 0,C 180,E1 -26746.739,E2 -26746.739} C_VEL
LIN {X 0,Y 103.72,Z 711.09,A -85,B 0,C 180,E1 -26752.934,E2 -26752.934} C_VEL
LIN {X 0,Y 105.027,Z 706.105,A -85,B 0,C 180,E1 -26756.855,E2 -26756.855} C_VEL
LIN {X 0,Y 106.897,Z 696.828,A -85,B 0,C 180,E1 -26762.851,E2 -26762.851} C_VEL
LIN {X 0,Y 109.319,Z 686.172,A -85,B 0,C 180,E1 -26768.231,E2 -26768.231} C_VEL
LIN {X 0,Y 111.584,Z 675.193,A -85,B 0,C 180,E1 -26772.624,E2 -26772.624} C_VEL
LIN {X 0,Y 113.523,Z 663.632,A -85,B 0,C 180,E1 -26776.352,E2 -26776.352} C_VEL
LIN {X 0,Y 114.834,Z 650.762,A -85,B 0,C 180,E1 -26779.825,E2 -26779.825} C_VEL
LIN {X 0,Y 114.846,Z 647.4,A -85,B 0,C 180,E1 -26780.7,E2 -26780.7} C_VEL
LIN {X 0,Y 111.456,Z 636.907,A -85,B 0,C 180,E1 -26784.871,E2 -26784.871} C_VEL
LIN {X 0,Y 109.822,Z 632.665,A -85,B 0,C 180,E1 -26786.703,E2 -26786.703} C_VEL
LIN {X 0,Y 107.932,Z 628.141,A -85,B 0,C 180,E1 -26788.741,E2 -26788.741} C_VEL
LIN {X 0,Y 105.763,Z 623.53,A -85,B 0,C 180,E1 -26791.062,E2 -26791.062} C_VEL
LIN {X 0,Y 105.073,Z 622.121,A -85,B 0,C 180,E1 -26791.809,E2 -26791.809} C_VEL
LIN {X 0,Y 102.467,Z 617.944,A -85,B 0,C 180,E1 -26794.592,E2 -26794.592} C_VEL
LIN {X 0,Y 101.564,Z 615.393,A -85,B 0,C 180,E1 -26795.875,E2 -26795.875} C_VEL
LIN {X 0,Y 100.893,Z 611.921,A -85,B 0,C 180,E1 -26802.909,E2 -26802.909} C_VEL
LIN {X 0,Y 101.206,Z 611.878,A -85,B 0,C 180,E1 -26807.974,E2 -26807.974} C_VEL
LIN {X 0,Y 101.285,Z 611.866,A -85,B 0,C 180,E1 -26812.021,E2 -26812.021} C_VEL
LIN {X 0,Y 101.875,Z 611.793,A -85,B 0,C 180,E1 -26819.998,E2 -26819.998} C_VEL
LIN {X 0,Y 101.258,Z 611.845,A -85,B 0,C 180,E1 -26826.66,E2 -26826.66} C_VEL
LIN {X 0,Y 100.903,Z 611.91,A -85,B 0,C 180,E1 -26828.874,E2 -26828.874} C_VEL
LIN {X 0,Y 99.438,Z 612.1,A -85,B 0,C 180,E1 -26832.151,E2 -26832.151} C_VEL
LIN {X 0,Y 93.935,Z 612.781,A -85,B 0,C 180,E1 -26842.425,E2 -26842.425} C_VEL
LIN {X 0,Y 93.643,Z 612.794,A -85,B 0,C 180,E1 -26844.894,E2 -26844.894} C_VEL
LIN {X 0,Y 93.656,Z 613.03,A -85,B 0,C 180,E1 -26852.52,E2 -26852.52} C_VEL
LIN {X 0,Y 94.778,Z 615.978,A -85,B 0,C 180,E1 -26855.099,E2 -26855.099} C_VEL
LIN {X 0,Y 97.39,Z 618.561,A -85,B 0,C 180,E1 -26859.1,E2 -26859.1} C_VEL
LIN {X 0,Y 98.367,Z 620.873,A -85,B 0,C 180,E1 -26860.925,E2 -26860.925} C_VEL
LIN {X 0,Y 100.053,Z 622.826,A -85,B 0,C 180,E1 -26863.223,E2 -26863.223} C_VEL
LIN {X 0,Y 102.758,Z 627.503,A -85,B 0,C 180,E1 -26867.182,E2 -26867.182} C_VEL
LIN {X 0,Y 106.225,Z 635.013,A -85,B 0,C 180,E1 -26872.553,E2 -26872.553} C_VEL
LIN {X 0,Y 108.845,Z 642.111,A -85,B 0,C 180,E1 -26877.073,E2 -26877.073} C_VEL
LIN {X 0,Y 110.847,Z 650.231,A -85,B 0,C 180,E1 -26881.861,E2 -26881.861} C_VEL
LIN {X 0,Y 111.743,Z 656.184,A -85,B 0,C 180,E1 -26885.337,E2 -26885.337} C_VEL
LIN {X 0,Y 111.74,Z 657.74,A -85,B 0,C 180,E1 -26886.171,E2 -26886.171} C_VEL
LIN {X 0,Y 108.053,Z 666.534,A -85,B 0,C 180,E1 -26890.03,E2 -26890.03} C_VEL
LIN {X 0,Y 103.886,Z 675.66,A -85,B 0,C 180,E1 -26895.3,E2 -26895.3} C_VEL
LIN {X 0,Y 100.326,Z 683.071,A -85,B 0,C 180,E1 -26900.928,E2 -26900.928} C_VEL
LIN {X 0,Y 98.026,Z 688.111,A -85,B 0,C 180,E1 -26905.885,E2 -26905.885} C_VEL
LIN {X 0,Y 96.038,Z 693.04,A -85,B 0,C 180,E1 -26912.093,E2 -26912.093} C_VEL
LIN {X 0,Y 94.973,Z 696.867,A -85,B 0,C 180,E1 -26918.507,E2 -26918.507} C_VEL
LIN {X 0,Y 95.083,Z 700.054,A -85,B 0,C 180,E1 -26926.083,E2 -26926.083} C_VEL
LIN {X 0,Y 96.014,Z 701.507,A -85,B 0,C 180,E1 -26931.464,E2 -26931.464} C_VEL
LIN {X 0,Y 97.232,Z 702.24,A -85,B 0,C 180,E1 -26935.697,E2 -26935.697} C_VEL
LIN {X 0,Y 100.657,Z 702.51,A -85,B 0,C 180,E1 -26943.088,E2 -26943.088} C_VEL
LIN {X 0,Y 103.612,Z 701.928,A -85,B 0,C 180,E1 -26947.619,E2 -26947.619} C_VEL
LIN {X 0,Y 107.273,Z 700.727,A -85,B 0,C 180,E1 -26952.112,E2 -26952.112} C_VEL
LIN {X 0,Y 106.737,Z 700.614,A -85,B 0,C 180,E1 -26953.593,E2 -26953.593} C_VEL
LIN {X 0,Y 99.165,Z 701.382,A -85,B 0,C 180,E1 -26961.216,E2 -26961.216} C_VEL
LIN {X 0,Y 94.918,Z 701.716,A -85,B 0,C 180,E1 -26968.939,E2 -26968.939} C_VEL
LIN {X 0,Y 93.342,Z 711.892,A -85,B 0,C 180,E1 -26974.614,E2 -26974.614} C_VEL
LIN {X 0,Y 92.268,Z 721.207,A -85,B 0,C 180,E1 -26981.114,E2 -26981.114} C_VEL
LIN {X 0,Y 91.859,Z 729.056,A -85,B 0,C 180,E1 -26987.856,E2 -26987.856} C_VEL
LIN {X 0,Y 92.56,Z 736.412,A -85,B 0,C 180,E1 -26995.647,E2 -26995.647} C_VEL
LIN {X 0,Y 95.084,Z 743.053,A -85,B 0,C 180,E1 -27004.241,E2 -27004.241} C_VEL
LIN {X 0,Y 99.656,Z 748.205,A -85,B 0,C 180,E1 -27012.216,E2 -27012.216} C_VEL
LIN {X 0,Y 106.128,Z 752.004,A -85,B 0,C 180,E1 -27019.338,E2 -27019.338} C_VEL
LIN {X 0,Y 114.3,Z 754.581,A -85,B 0,C 180,E1 -27025.495,E2 -27025.495} C_VEL
LIN {X 0,Y 123.89,Z 755.979,A -85,B 0,C 180,E1 -27030.702,E2 -27030.702} C_VEL
LIN {X 0,Y 134.69,Z 756.158,A -85,B 0,C 180,E1 -27035.029,E2 -27035.029} C_VEL
LIN {X 0,Y 138.117,Z 755.943,A -85,B 0,C 180,E1 -27036.187,E2 -27036.187} C_VEL
LIN {X 0,Y 136.386,Z 756.365,A -85,B 0,C 180,E1 -27037.471,E2 -27037.471} C_VEL
LIN {X 0,Y 128.772,Z 757.41,A -85,B 0,C 180,E1 -27040.18,E2 -27040.18} C_VEL
LIN {X 0,Y 118.769,Z 758.006,A -85,B 0,C 180,E1 -27044.763,E2 -27044.763} C_VEL
LIN {X 0,Y 110.013,Z 757.588,A -85,B 0,C 180,E1 -27050.3,E2 -27050.3} C_VEL
LIN {X 0,Y 102.855,Z 756.159,A -85,B 0,C 180,E1 -27056.868,E2 -27056.868} C_VEL
LIN {X 0,Y 97.556,Z 753.694,A -85,B 0,C 180,E1 -27064.394,E2 -27064.394} C_VEL
LIN {X 0,Y 94.557,Z 750.095,A -85,B 0,C 180,E1 -27072.709,E2 -27072.709} C_VEL
LIN {X 0,Y 93.858,Z 745.233,A -85,B 0,C 180,E1 -27081.391,E2 -27081.391} C_VEL
LIN {X 0,Y 94.226,Z 742.211,A -85,B 0,C 180,E1 -27085.727,E2 -27085.727} C_VEL
LIN {X 0,Y 94.169,Z 738.434,A -85,B 0,C 180,E1 -27090.004,E2 -27090.004} C_VEL
LIN {X 0,Y 94.025,Z 732.533,A -85,B 0,C 180,E1 -27095.365,E2 -27095.365} C_VEL
LIN {X 0,Y 94.385,Z 723.709,A -85,B 0,C 180,E1 -27101.82,E2 -27101.82} C_VEL
LIN {X 0,Y 94.988,Z 718.267,A -85,B 0,C 180,E1 -27105.27,E2 -27105.27} C_VEL
LIN {X 0,Y 96.375,Z 711.786,A -85,B 0,C 180,E1 -27112.514,E2 -27112.514} C_VEL
LIN {X 0,Y 97.834,Z 707.122,A -85,B 0,C 180,E1 -27116.682,E2 -27116.682} C_VEL
LIN {X 0,Y 99.896,Z 697.801,A -85,B 0,C 180,E1 -27123.459,E2 -27123.459} C_VEL
LIN {X 0,Y 102.303,Z 688.363,A -85,B 0,C 180,E1 -27128.824,E2 -27128.824} C_VEL
LIN {X 0,Y 104.841,Z 678.163,A -85,B 0,C 180,E1 -27133.406,E2 -27133.406} C_VEL
LIN {X 0,Y 107.212,Z 666.61,A -85,B 0,C 180,E1 -27137.621,E2 -27137.621} C_VEL
LIN {X 0,Y 108.933,Z 654.585,A -85,B 0,C 180,E1 -27141.266,E2 -27141.266} C_VEL
LIN {X 0,Y 109.285,Z 650.624,A -85,B 0,C 180,E1 -27142.339,E2 -27142.339} C_VEL
LIN {X 0,Y 106.942,Z 641.999,A -85,B 0,C 180,E1 -27146.074,E2 -27146.074} C_VEL
LIN {X 0,Y 103.738,Z 632.963,A -85,B 0,C 180,E1 -27150.441,E2 -27150.441} C_VEL
LIN {X 0,Y 101.225,Z 627.19,A -85,B 0,C 180,E1 -27153.727,E2 -27153.727} C_VEL
LIN {X 0,Y 98.8,Z 622.458,A -85,B 0,C 180,E1 -27156.967,E2 -27156.967} C_VEL
LIN {X 0,Y 98.079,Z 620.78,A -85,B 0,C 180,E1 -27158.038,E2 -27158.038} C_VEL
LIN {X 0,Y 94.975,Z 615.988,A -85,B 0,C 180,E1 -27162.642,E2 -27162.642} C_VEL
LIN {X 0,Y 93.993,Z 613.119,A -85,B 0,C 180,E1 -27164.765,E2 -27164.765} C_VEL
LIN {X 0,Y 94.054,Z 612.774,A -85,B 0,C 180,E1 -27166.279,E2 -27166.279} C_VEL
LIN {X 0,Y 94.218,Z 612.747,A -85,B 0,C 180,E1 -27171.418,E2 -27171.418} C_VEL
LIN {X 0,Y 94.801,Z 612.674,A -85,B 0,C 180,E1 -27179.998,E2 -27179.998} C_VEL
LIN {X 0,Y 94.21,Z 612.74,A -85,B 0,C 180,E1 -27188.579,E2 -27188.579} C_VEL
LIN {X 0,Y 94.051,Z 612.745,A -85,B 0,C 180,E1 -27193.713,E2 -27193.713} C_VEL
LIN {X 0,Y 93.699,Z 612.813,A -85,B 0,C 180,E1 -27202.024,E2 -27202.024} C_VEL
LIN {X 0,Y 93.643,Z 612.794,A -85,B 0,C 180,E1 -27204.894,E2 -27204.894} C_VEL
LIN {X 0,Y 93.653,Z 613.31,A -85,B 0,C 180,E1 -27207.249,E2 -27207.249} C_VEL
LIN {X 0,Y 93.62,Z 615.568,A -85,B 0,C 180,E1 -27210.574,E2 -27210.574} C_VEL
LIN {X 0,Y 93.677,Z 618.863,A -85,B 0,C 180,E1 -27213.621,E2 -27213.621} C_VEL
LIN {X 0,Y 94.915,Z 626.314,A -85,B 0,C 180,E1 -27219.593,E2 -27219.593} C_VEL
LIN {X 0,Y 95.99,Z 628.304,A -85,B 0,C 180,E1 -27221.65,E2 -27221.65} C_VEL
LIN {X 0,Y 98.314,Z 632.347,A -85,B 0,C 180,E1 -27225.629,E2 -27225.629} C_VEL
LIN {X 0,Y 101.323,Z 639.67,A -85,B 0,C 180,E1 -27231.368,E2 -27231.368} C_VEL
LIN {X 0,Y 103.539,Z 646.635,A -85,B 0,C 180,E1 -27236.25,E2 -27236.25} C_VEL
LIN {X 0,Y 105.002,Z 653.92,A -85,B 0,C 180,E1 -27240.983,E2 -27240.983} C_VEL
LIN {X 0,Y 105.553,Z 658.699,A -85,B 0,C 180,E1 -27244.019,E2 -27244.019} C_VEL
LIN {X 0,Y 105.419,Z 659.743,A -85,B 0,C 180,E1 -27244.578,E2 -27244.578} C_VEL
LIN {X 0,Y 101.43,Z 668.452,A -85,B 0,C 180,E1 -27248.664,E2 -27248.664} C_VEL
LIN {X 0,Y 97.058,Z 677.413,A -85,B 0,C 180,E1 -27254.24,E2 -27254.24} C_VEL
LIN {X 0,Y 93.332,Z 684.697,A -85,B 0,C 180,E1 -27260.242,E2 -27260.242} C_VEL
LIN {X 0,Y 90.935,Z 689.626,A -85,B 0,C 180,E1 -27265.563,E2 -27265.563} C_VEL
LIN {X 0,Y 88.879,Z 694.461,A -85,B 0,C 180,E1 -27272.262,E2 -27272.262} C_VEL
LIN {X 0,Y 87.871,Z 698.193,A -85,B 0,C 180,E1 -27279.2,E2 -27279.2} C_VEL
LIN {X 0,Y 88.098,Z 701.098,A -85,B 0,C 180,E1 -27286.81,E2 -27286.81} C_VEL
LIN {X 0,Y 89.323,Z 702.656,A -85,B 0,C 180,E1 -27293.162,E2 -27293.162} C_VEL
LIN {X 0,Y 90.762,Z 703.345,A -85,B 0,C 180,E1 -27297.679,E2 -27297.679} C_VEL
LIN {X 0,Y 94.393,Z 703.522,A -85,B 0,C 180,E1 -27305.018,E2 -27305.018} C_VEL
LIN {X 0,Y 99.013,Z 702.568,A -85,B 0,C 180,E1 -27311.557,E2 -27311.557} C_VEL
LIN {X 0,Y 97.873,Z 702.598,A -85,B 0,C 180,E1 -27314.107,E2 -27314.107} C_VEL
LIN {X 0,Y 91.291,Z 703.432,A -85,B 0,C 180,E1 -27321.987,E2 -27321.987} C_VEL
LIN {X 0,Y 87.427,Z 703.86,A -85,B 0,C 180,E1 -27329.842,E2 -27329.842} C_VEL
LIN {X 0,Y 87.316,Z 704.057,A -85,B 0,C 180,E1 -27330.795,E2 -27330.795} C_VEL
LIN {X 0,Y 85.918,Z 714.033,A -85,B 0,C 180,E1 -27337.138,E2 -27337.138} C_VEL
LIN {X 0,Y 85.12,Z 723.255,A -85,B 0,C 180,E1 -27344.437,E2 -27344.437} C_VEL
LIN {X 0,Y 85.156,Z 730.909,A -85,B 0,C 180,E1 -27352.008,E2 -27352.008} C_VEL
LIN {X 0,Y 86.565,Z 737.675,A -85,B 0,C 180,E1 -27360.002,E2 -27360.002} C_VEL
LIN {X 0,Y 90.088,Z 744.092,A -85,B 0,C 180,E1 -27368.978,E2 -27368.978} C_VEL
LIN {X 0,Y 95.757,Z 749.065,A -85,B 0,C 180,E1 -27377.074,E2 -27377.074} C_VEL
LIN {X 0,Y 103.35,Z 752.756,A -85,B 0,C 180,E1 -27384.082,E2 -27384.082} C_VEL
LIN {X 0,Y 112.59,Z 755.29,A -85,B 0,C 180,E1 -27389.96,E2 -27389.96} C_VEL
LIN {X 0,Y 123.081,Z 756.638,A -85,B 0,C 180,E1 -27394.822,E2 -27394.822} C_VEL
LIN {X 0,Y 126.497,Z 756.798,A -85,B 0,C 180,E1 -27396.11,E2 -27396.11} C_VEL
LIN {X 0,Y 125.655,Z 756.993,A -85,B 0,C 180,E1 -27397.195,E2 -27397.195} C_VEL
LIN {X 0,Y 113.914,Z 757.303,A -85,B 0,C 180,E1 -27402.244,E2 -27402.244} C_VEL
LIN {X 0,Y 104.702,Z 756.517,A -85,B 0,C 180,E1 -27407.843,E2 -27407.843} C_VEL
LIN {X 0,Y 97.076,Z 754.771,A -85,B 0,C 180,E1 -27414.613,E2 -27414.613} C_VEL
LIN {X 0,Y 91.377,Z 751.971,A -85,B 0,C 180,E1 -27422.523,E2 -27422.523} C_VEL
LIN {X 0,Y 88.058,Z 748.088,A -85,B 0,C 180,E1 -27431.387,E2 -27431.387} C_VEL
LIN {X 0,Y 87.216,Z 742.949,A -85,B 0,C 180,E1 -27440.73,E2 -27440.73} C_VEL
LIN {X 0,Y 87.571,Z 739.723,A -85,B 0,C 180,E1 -27445.401,E2 -27445.401} C_VEL
LIN {X 0,Y 87.464,Z 735.655,A -85,B 0,C 180,E1 -27450.004,E2 -27450.004} C_VEL
LIN {X 0,Y 87.232,Z 727.985,A -85,B 0,C 180,E1 -27456.945,E2 -27456.945} C_VEL
LIN {X 0,Y 87.854,Z 718.632,A -85,B 0,C 180,E1 -27463.89,E2 -27463.89} C_VEL
LIN {X 0,Y 88.735,Z 713.401,A -85,B 0,C 180,E1 -27470.884,E2 -27470.884} C_VEL
LIN {X 0,Y 90.888,Z 706.789,A -85,B 0,C 180,E1 -27477.647,E2 -27477.647} C_VEL
LIN {X 0,Y 92.782,Z 699.097,A -85,B 0,C 180,E1 -27483.869,E2 -27483.869} C_VEL
LIN {X 0,Y 95.582,Z 689.343,A -85,B 0,C 180,E1 -27490.048,E2 -27490.048} C_VEL
LIN {X 0,Y 98.154,Z 680.419,A -85,B 0,C 180,E1 -27494.527,E2 -27494.527} C_VEL
LIN {X 0,Y 100.96,Z 668.979,A -85,B 0,C 180,E1 -27499.208,E2 -27499.208} C_VEL
LIN {X 0,Y 102.969,Z 658.375,A -85,B 0,C 180,E1 -27502.768,E2 -27502.768} C_VEL
LIN {X 0,Y 103.608,Z 654.083,A -85,B 0,C 180,E1 -27504.046,E2 -27504.046} C_VEL
LIN {X 0,Y 103.051,Z 650.402,A -85,B 0,C 180,E1 -27505.635,E2 -27505.635} C_VEL
LIN {X 0,Y 100.929,Z 642.319,A -85,B 0,C 180,E1 -27509.678,E2 -27509.678} C_VEL
LIN {X 0,Y 99.195,Z 637.136,A -85,B 0,C 180,E1 -27512.577,E2 -27512.577} C_VEL
LIN {X 0,Y 97.434,Z 632.433,A -85,B 0,C 180,E1 -27515.494,E2 -27515.494} C_VEL
LIN {X 0,Y 95.254,Z 627.305,A -85,B 0,C 180,E1 -27519.2,E2 -27519.2} C_VEL
LIN {X 0,Y 94.184,Z 625.461,A -85,B 0,C 180,E1 -27520.944,E2 -27520.944} C_VEL
LIN {X 0,Y 91.861,Z 620.592,A -85,B 0,C 180,E1 -27525.576,E2 -27525.576} C_VEL
LIN {X 0,Y 91.411,Z 619.35,A -85,B 0,C 180,E1 -27526.663,E2 -27526.663} C_VEL
LIN {X 0,Y 88.855,Z 617.419,A -85,B 0,C 180,E1 -27532.042,E2 -27532.042} C_VEL
LIN {X 0,Y 87.612,Z 614.941,A -85,B 0,C 180,E1 -27536.405,E2 -27536.405} C_VEL
LIN {X 0,Y 87.457,Z 613.589,A -85,B 0,C 180,E1 -27537.983,E2 -27537.983} C_VEL
LIN {X 0,Y 87.728,Z 613.554,A -85,B 0,C 180,E1 -27539.998,E2 -27539.998} C_VEL
LIN {X 0,Y 87.118,Z 613.629,A -85,B 0,C 180,E1 -27549.283,E2 -27549.283} C_VEL
LIN {X 0,Y 86.956,Z 613.625,A -85,B 0,C 180,E1 -27554.085,E2 -27554.085} C_VEL
LIN {X 0,Y 86.779,Z 613.83,A -85,B 0,C 180,E1 -27557.373,E2 -27557.373} C_VEL
LIN {X 0,Y 87.261,Z 615.807,A -85,B 0,C 180,E1 -27560.938,E2 -27560.938} C_VEL
LIN {X 0,Y 89.969,Z 618.946,A -85,B 0,C 180,E1 -27569.223,E2 -27569.223} C_VEL
LIN {X 0,Y 90.955,Z 619.644,A -85,B 0,C 180,E1 -27571.276,E2 -27571.276} C_VEL
LIN {X 0,Y 91.871,Z 622.128,A -85,B 0,C 180,E1 -27573.85,E2 -27573.85} C_VEL
LIN {X 0,Y 94.104,Z 624.86,A -85,B 0,C 180,E1 -27578.032,E2 -27578.032} C_VEL
LIN {X 0,Y 95.99,Z 628.304,A -85,B 0,C 180,E1 -27581.65,E2 -27581.65} C_VEL
LIN {X 0,Y 97.067,Z 630.287,A -85,B 0,C 180,E1 -27583.557,E2 -27583.557} C_VEL
LIN {X 0,Y 97.96,Z 634.145,A -85,B 0,C 180,E1 -27586.145,E2 -27586.145} C_VEL
LIN {X 0,Y 98.191,Z 638.555,A -85,B 0,C 180,E1 -27588.491,E2 -27588.491} C_VEL
LIN {X 0,Y 97.891,Z 647.786,A -85,B 0,C 180,E1 -27593.266,E2 -27593.266} C_VEL
LIN {X 0,Y 98.06,Z 650.56,A -85,B 0,C 180,E1 -27595.028,E2 -27595.028} C_VEL
LIN {X 0,Y 99.155,Z 657.898,A -85,B 0,C 180,E1 -27600.25,E2 -27600.25} C_VEL
LIN {X 0,Y 99.321,Z 659.802,A -85,B 0,C 180,E1 -27601.58,E2 -27601.58} C_VEL
LIN {X 0,Y 99.139,Z 661.724,A -85,B 0,C 180,E1 -27602.786,E2 -27602.786} C_VEL
LIN {X 0,Y 94.064,Z 671.975,A -85,B 0,C 180,E1 -27608.06,E2 -27608.06} C_VEL
LIN {X 0,Y 89.57,Z 680.445,A -85,B 0,C 180,E1 -27614.056,E2 -27614.056} C_VEL
LIN {X 0,Y 85.779,Z 687.311,A -85,B 0,C 180,E1 -27620.565,E2 -27620.565} C_VEL
LIN {X 0,Y 83.002,Z 692.827,A -85,B 0,C 180,E1 -27627.569,E2 -27627.569} C_VEL
LIN {X 0,Y 81.281,Z 697.181,A -85,B 0,C 180,E1 -27634.956,E2 -27634.956} C_VEL
LIN {X 0,Y 80.789,Z 699.515,A -85,B 0,C 180,E1 -27640.015,E2 -27640.015} C_VEL
LIN {X 0,Y 81.142,Z 702.15,A -85,B 0,C 180,E1 -27647.689,E2 -27647.689} C_VEL
LIN {X 0,Y 82.711,Z 703.808,A -85,B 0,C 180,E1 -27655.136,E2 -27655.136} C_VEL
LIN {X 0,Y 84.43,Z 704.418,A -85,B 0,C 180,E1 -27659.958,E2 -27659.958} C_VEL
LIN {X 0,Y 89.381,Z 704.392,A -85,B 0,C 180,E1 -27668.973,E2 -27668.973} C_VEL
LIN {X 0,Y 90.803,Z 704.153,A -85,B 0,C 180,E1 -27670.941,E2 -27670.941} C_VEL
LIN {X 0,Y 91.283,Z 704.031,A -85,B 0,C 180,E1 -27672.542,E2 -27672.542} C_VEL
LIN {X 0,Y 80.835,Z 705.74,A -85,B 0,C 180,E1 -27688.559,E2 -27688.559} C_VEL
LIN {X 0,Y 79.849,Z 705.969,A -85,B 0,C 180,E1 -27692.823,E2 -27692.823} C_VEL
LIN {X 0,Y 78.755,Z 714.768,A -85,B 0,C 180,E1 -27699.089,E2 -27699.089} C_VEL
LIN {X 0,Y 78.176,Z 723.666,A -85,B 0,C 180,E1 -27707.014,E2 -27707.014} C_VEL
LIN {X 0,Y 78.601,Z 730.964,A -85,B 0,C 180,E1 -27714.872,E2 -27714.872} C_VEL
LIN {X 0,Y 80.229,Z 737.027,A -85,B 0,C 180,E1 -27722.512,E2 -27722.512} C_VEL
LIN {X 0,Y 84.392,Z 743.587,A -85,B 0,C 180,E1 -27732.019,E2 -27732.019} C_VEL
LIN {X 0,Y 90.775,Z 748.768,A -85,B 0,C 180,E1 -27740.391,E2 -27740.391} C_VEL
LIN {X 0,Y 96.806,Z 751.817,A -85,B 0,C 180,E1 -27745.825,E2 -27745.825} C_VEL
LIN {X 0,Y 106.345,Z 754.865,A -85,B 0,C 180,E1 -27751.919,E2 -27751.919} C_VEL
LIN {X 0,Y 115.089,Z 756.508,A -85,B 0,C 180,E1 -27756.031,E2 -27756.031} C_VEL
LIN {X 0,Y 114.594,Z 756.641,A -85,B 0,C 180,E1 -27757.135,E2 -27757.135} C_VEL
LIN {X 0,Y 101.586,Z 755.617,A -85,B 0,C 180,E1 -27763.777,E2 -27763.777} C_VEL
LIN {X 0,Y 91.519,Z 753.193,A -85,B 0,C 180,E1 -27772.101,E2 -27772.101} C_VEL
LIN {X 0,Y 85.359,Z 750.083,A -85,B 0,C 180,E1 -27780.401,E2 -27780.401} C_VEL
LIN {X 0,Y 81.687,Z 745.928,A -85,B 0,C 180,E1 -27789.876,E2 -27789.876} C_VEL
LIN {X 0,Y 80.673,Z 740.449,A -85,B 0,C 180,E1 -27799.971,E2 -27799.971} C_VEL
LIN {X 0,Y 80.962,Z 737.102,A -85,B 0,C 180,E1 -27805.025,E2 -27805.025} C_VEL
LIN {X 0,Y 80.749,Z 732.735,A -85,B 0,C 180,E1 -27810.005,E2 -27810.005} C_VEL
LIN {X 0,Y 80.468,Z 725.994,A -85,B 0,C 180,E1 -27816.272,E2 -27816.272} C_VEL
LIN {X 0,Y 80.75,Z 719.342,A -85,B 0,C 180,E1 -27821.616,E2 -27821.616} C_VEL
LIN {X 0,Y 81.478,Z 713.862,A -85,B 0,C 180,E1 -27830.188,E2 -27830.188} C_VEL
LIN {X 0,Y 83.641,Z 707.613,A -85,B 0,C 180,E1 -27837.53,E2 -27837.53} C_VEL
LIN {X 0,Y 85.997,Z 699.225,A -85,B 0,C 180,E1 -27845.188,E2 -27845.188} C_VEL
LIN {X 0,Y 88.608,Z 691.225,A -85,B 0,C 180,E1 -27850.876,E2 -27850.876} C_VEL
LIN {X 0,Y 91.914,Z 681.113,A -85,B 0,C 180,E1 -27856.513,E2 -27856.513} C_VEL
LIN {X 0,Y 95.218,Z 669.389,A -85,B 0,C 180,E1 -27861.655,E2 -27861.655} C_VEL
LIN {X 0,Y 97.734,Z 658.011,A -85,B 0,C 180,E1 -27865.723,E2 -27865.723} C_VEL
LIN {X 0,Y 98.042,Z 656.324,A -85,B 0,C 180,E1 -27866.25,E2 -27866.25} C_VEL
LIN {X 0,Y 96.736,Z 649.04,A -85,B 0,C 180,E1 -27870.092,E2 -27870.092} C_VEL
LIN {X 0,Y 95.215,Z 642.852,A -85,B 0,C 180,E1 -27873.711,E2 -27873.711} C_VEL
LIN {X 0,Y 93.804,Z 638.089,A -85,B 0,C 180,E1 -27876.836,E2 -27876.836} C_VEL
LIN {X 0,Y 91.323,Z 631.707,A -85,B 0,C 180,E1 -27882.07,E2 -27882.07} C_VEL
LIN {X 0,Y 89.227,Z 626.706,A -85,B 0,C 180,E1 -27887.199,E2 -27887.199} C_VEL
LIN {X 0,Y 88.963,Z 625.853,A -85,B 0,C 180,E1 -27888.03,E2 -27888.03} C_VEL
LIN {X 0,Y 86.492,Z 623.568,A -85,B 0,C 180,E1 -27894.169,E2 -27894.169} C_VEL
LIN {X 0,Y 85.643,Z 620.828,A -85,B 0,C 180,E1 -27898.676,E2 -27898.676} C_VEL
LIN {X 0,Y 85.442,Z 620.256,A -85,B 0,C 180,E1 -27899.998,E2 -27899.998} C_VEL
LIN {X 0,Y 84.843,Z 620.449,A -85,B 0,C 180,E1 -27915.616,E2 -27915.616} C_VEL
LIN {X 0,Y 86.041,Z 624.06,A -85,B 0,C 180,E1 -27924.103,E2 -27924.103} C_VEL
LIN {X 0,Y 87.566,Z 625.581,A -85,B 0,C 180,E1 -27928.785,E2 -27928.785} C_VEL
LIN {X 0,Y 89.1,Z 628.801,A -85,B 0,C 180,E1 -27933.512,E2 -27933.512} C_VEL
LIN {X 0,Y 90.134,Z 630.079,A -85,B 0,C 180,E1 -27935.786,E2 -27935.786} C_VEL
LIN {X 0,Y 92.63,Z 634.716,A -85,B 0,C 180,E1 -27941.428,E2 -27941.428} C_VEL
LIN {X 0,Y 95.298,Z 641.127,A -85,B 0,C 180,E1 -27947.514,E2 -27947.514} C_VEL
LIN {X 0,Y 97.266,Z 647.439,A -85,B 0,C 180,E1 -27952.635,E2 -27952.635} C_VEL
LIN {X 0,Y 98.06,Z 650.56,A -85,B 0,C 180,E1 -27955.028,E2 -27955.028} C_VEL
LIN {X 0,Y 97.907,Z 653.393,A -85,B 0,C 180,E1 -27956.64,E2 -27956.64} C_VEL
LIN {X 0,Y 96.958,Z 656.456,A -85,B 0,C 180,E1 -27958.001,E2 -27958.001} C_VEL
LIN {X 0,Y 91.365,Z 666.839,A -85,B 0,C 180,E1 -27962.294,E2 -27962.294} C_VEL
LIN {X 0,Y 86.712,Z 675.326,A -85,B 0,C 180,E1 -27967.353,E2 -27967.353} C_VEL
LIN {X 0,Y 82.029,Z 683.383,A -85,B 0,C 180,E1 -27973.828,E2 -27973.828} C_VEL
LIN {X 0,Y 78.338,Z 689.685,A -85,B 0,C 180,E1 -27980.686,E2 -27980.686} C_VEL
LIN {X 0,Y 75.848,Z 694.299,A -85,B 0,C 180,E1 -27987.34,E2 -27987.34} C_VEL
LIN {X 0,Y 74.152,Z 698.551,A -85,B 0,C 180,E1 -27995.433,E2 -27995.433} C_VEL
LIN {X 0,Y 73.724,Z 700.803,A -85,B 0,C 180,E1 -28000.986,E2 -28000.986} C_VEL
LIN {X 0,Y 74.233,Z 703.213,A -85,B 0,C 180,E1 -28008.788,E2 -28008.788} C_VEL
LIN {X 0,Y 76.235,Z 704.946,A -85,B 0,C 180,E1 -28017.442,E2 -28017.442} C_VEL
LIN {X 0,Y 80.795,Z 705.62,A -85,B 0,C 180,E1 -28027.504,E2 -28027.504} C_VEL
LIN {X 0,Y 82.197,Z 705.555,A -85,B 0,C 180,E1 -28029.693,E2 -28029.693} C_VEL
LIN {X 0,Y 82.772,Z 705.566,A -85,B 0,C 180,E1 -28032.78,E2 -28032.78} C_VEL
LIN {X 0,Y 73.064,Z 707.633,A -85,B 0,C 180,E1 -28051.255,E2 -28051.255} C_VEL
LIN {X 0,Y 72.506,Z 707.963,A -85,B 0,C 180,E1 -28055.484,E2 -28055.484} C_VEL
LIN {X 0,Y 71.594,Z 716.818,A -85,B 0,C 180,E1 -28062.875,E2 -28062.875} C_VEL
LIN {X 0,Y 71.537,Z 725.716,A -85,B 0,C 180,E1 -28071.951,E2 -28071.951} C_VEL
LIN {X 0,Y 72.939,Z 733.29,A -85,B 0,C 180,E1 -28081.382,E2 -28081.382} C_VEL
LIN {X 0,Y 76.24,Z 739.846,A -85,B 0,C 180,E1 -28090.626,E2 -28090.626} C_VEL
LIN {X 0,Y 82.292,Z 745.852,A -85,B 0,C 180,E1 -28099.977,E2 -28099.977} C_VEL
LIN {X 0,Y 90.391,Z 750.599,A -85,B 0,C 180,E1 -28107.81,E2 -28107.81} C_VEL
LIN {X 0,Y 100.244,Z 754.169,A -85,B 0,C 180,E1 -28114.118,E2 -28114.118} C_VEL
LIN {X 0,Y 104.968,Z 755.398,A -85,B 0,C 180,E1 -28116.546,E2 -28116.546} C_VEL
LIN {X 0,Y 94.813,Z 753.898,A -85,B 0,C 180,E1 -28122.168,E2 -28122.168} C_VEL
LIN {X 0,Y 86.187,Z 751.482,A -85,B 0,C 180,E1 -28129.287,E2 -28129.287} C_VEL
LIN {X 0,Y 79.491,Z 748.072,A -85,B 0,C 180,E1 -28137.968,E2 -28137.968} C_VEL
LIN {X 0,Y 75.145,Z 743.002,A -85,B 0,C 180,E1 -28149.276,E2 -28149.276} C_VEL
LIN {X 0,Y 74.2,Z 737.79,A -85,B 0,C 180,E1 -28159.085,E2 -28159.085} C_VEL
LIN {X 0,Y 74.423,Z 734.224,A -85,B 0,C 180,E1 -28164.586,E2 -28164.586} C_VEL
LIN {X 0,Y 74.057,Z 729.577,A -85,B 0,C 180,E1 -28170.005,E2 -28170.005} C_VEL
LIN {X 0,Y 73.761,Z 722.462,A -85,B 0,C 180,E1 -28176.845,E2 -28176.845} C_VEL
LIN {X 0,Y 73.83,Z 719.705,A -85,B 0,C 180,E1 -28179.249,E2 -28179.249} C_VEL
LIN {X 0,Y 74.232,Z 714.107,A -85,B 0,C 180,E1 -28189.555,E2 -28189.555} C_VEL
LIN {X 0,Y 76.24,Z 708.345,A -85,B 0,C 180,E1 -28197.451,E2 -28197.451} C_VEL
LIN {X 0,Y 77.841,Z 703.465,A -85,B 0,C 180,E1 -28202.806,E2 -28202.806} C_VEL
LIN {X 0,Y 80.998,Z 694.565,A -85,B 0,C 180,E1 -28210.604,E2 -28210.604} C_VEL
LIN {X 0,Y 84.451,Z 685.38,A -85,B 0,C 180,E1 -28216.739,E2 -28216.739} C_VEL
LIN {X 0,Y 88.053,Z 674.914,A -85,B 0,C 180,E1 -28222.166,E2 -28222.166} C_VEL
LIN {X 0,Y 91.348,Z 663.704,A -85,B 0,C 180,E1 -28226.799,E2 -28226.799} C_VEL
LIN {X 0,Y 92.54,Z 658.253,A -85,B 0,C 180,E1 -28228.843,E2 -28228.843} C_VEL
LIN {X 0,Y 91.292,Z 650.285,A -85,B 0,C 180,E1 -28233.724,E2 -28233.724} C_VEL
LIN {X 0,Y 89.851,Z 643.875,A -85,B 0,C 180,E1 -28238.188,E2 -28238.188} C_VEL
LIN {X 0,Y 88.253,Z 638.237,A -85,B 0,C 180,E1 -28242.879,E2 -28242.879} C_VEL
LIN {X 0,Y 86.432,Z 633.318,A -85,B 0,C 180,E1 -28248.269,E2 -28248.269} C_VEL
LIN {X 0,Y 85.669,Z 631.885,A -85,B 0,C 180,E1 -28250.555,E2 -28250.555} C_VEL
LIN {X 0,Y 83.724,Z 628.922,A -85,B 0,C 180,E1 -28257.593,E2 -28257.593} C_VEL
LIN {X 0,Y 83.451,Z 627.105,A -85,B 0,C 180,E1 -28260.602,E2 -28260.602} C_VEL
LIN {X 0,Y 82.705,Z 627.188,A -85,B 0,C 180,E1 -28274.767,E2 -28274.767} C_VEL
LIN {X 0,Y 85.124,Z 633.013,A -85,B 0,C 180,E1 -28289.692,E2 -28289.692} C_VEL
LIN {X 0,Y 85.713,Z 634.713,A -85,B 0,C 180,E1 -28292.204,E2 -28292.204} C_VEL
LIN {X 0,Y 86.598,Z 635.971,A -85,B 0,C 180,E1 -28294.615,E2 -28294.615} C_VEL
LIN {X 0,Y 89.07,Z 641.602,A -85,B 0,C 180,E1 -28301.771,E2 -28301.771} C_VEL
LIN {X 0,Y 90.852,Z 647.096,A -85,B 0,C 180,E1 -28307.292,E2 -28307.292} C_VEL
LIN {X 0,Y 92.292,Z 652.985,A -85,B 0,C 180,E1 -28312.464,E2 -28312.464} C_VEL
LIN {X 0,Y 93.156,Z 660.053,A -85,B 0,C 180,E1 -28318.118,E2 -28318.118} C_VEL
LIN {X 0,Y 93.257,Z 661.897,A -85,B 0,C 180,E1 -28319.527,E2 -28319.527} C_VEL
LIN {X 0,Y 92.96,Z 663.74,A -85,B 0,C 180,E1 -28320.776,E2 -28320.776} C_VEL
LIN {X 0,Y 91.365,Z 666.839,A -85,B 0,C 180,E1 -28322.294,E2 -28322.294} C_VEL
LIN {X 0,Y 88.651,Z 671.034,A -85,B 0,C 180,E1 -28324.326,E2 -28324.326} C_VEL
LIN {X 0,Y 82.769,Z 677.553,A -85,B 0,C 180,E1 -28327.403,E2 -28327.403} C_VEL
LIN {X 0,Y 76.778,Z 683.535,A -85,B 0,C 180,E1 -28331.153,E2 -28331.153} C_VEL
LIN {X 0,Y 74.035,Z 686.834,A -85,B 0,C 180,E1 -28334.244,E2 -28334.244} C_VEL
LIN {X 0,Y 70.748,Z 692.149,A -85,B 0,C 180,E1 -28341.137,E2 -28341.137} C_VEL
LIN {X 0,Y 67.962,Z 697.249,A -85,B 0,C 180,E1 -28349.995,E2 -28349.995} C_VEL
LIN {X 0,Y 66.738,Z 701.048,A -85,B 0,C 180,E1 -28359.083,E2 -28359.083} C_VEL
LIN {X 0,Y 67.363,Z 704.278,A -85,B 0,C 180,E1 -28370.128,E2 -28370.128} C_VEL
LIN {X 0,Y 69.881,Z 706.056,A -85,B 0,C 180,E1 -28380.182,E2 -28380.182} C_VEL
LIN {X 0,Y 75.191,Z 706.636,A -85,B 0,C 180,E1 -28390.858,E2 -28390.858} C_VEL
LIN {X 0,Y 75.36,Z 706.685,A -85,B 0,C 180,E1 -28391.752,E2 -28391.752} C_VEL
LIN {X 0,Y 66.674,Z 708.835,A -85,B 0,C 180,E1 -28408.197,E2 -28408.197} C_VEL
LIN {X 0,Y 65.179,Z 709.839,A -85,B 0,C 180,E1 -28418.869,E2 -28418.869} C_VEL
LIN {X 0,Y 64.678,Z 718.711,A -85,B 0,C 180,E1 -28427.451,E2 -28427.451} C_VEL
LIN {X 0,Y 65.248,Z 726.697,A -85,B 0,C 180,E1 -28436.915,E2 -28436.915} C_VEL
LIN {X 0,Y 67.249,Z 733.393,A -85,B 0,C 180,E1 -28446.001,E2 -28446.001} C_VEL
LIN {X 0,Y 72.269,Z 740.714,A -85,B 0,C 180,E1 -28456.965,E2 -28456.965} C_VEL
LIN {X 0,Y 79.681,Z 746.617,A -85,B 0,C 180,E1 -28466.171,E2 -28466.171} C_VEL
LIN {X 0,Y 89.038,Z 751.269,A -85,B 0,C 180,E1 -28473.543,E2 -28473.543} C_VEL
LIN {X 0,Y 93.618,Z 753.051,A -85,B 0,C 180,E1 -28476.912,E2 -28476.912} C_VEL
LIN {X 0,Y 85.474,Z 751.091,A -85,B 0,C 180,E1 -28482.274,E2 -28482.274} C_VEL
LIN {X 0,Y 77.164,Z 747.855,A -85,B 0,C 180,E1 -28490.397,E2 -28490.397} C_VEL
LIN {X 0,Y 70.173,Z 742.391,A -85,B 0,C 180,E1 -28503.222,E2 -28503.222} C_VEL
LIN {X 0,Y 67.878,Z 736.644,A -85,B 0,C 180,E1 -28515.004,E2 -28515.004} C_VEL
LIN {X 0,Y 67.927,Z 732.233,A -85,B 0,C 180,E1 -28522.575,E2 -28522.575} C_VEL
LIN {X 0,Y 67.662,Z 728.792,A -85,B 0,C 180,E1 -28527.029,E2 -28527.029} C_VEL
LIN {X 0,Y 67.102,Z 721.746,A -85,B 0,C 180,E1 -28534.511,E2 -28534.511} C_VEL
LIN {X 0,Y 67.039,Z 719.906,A -85,B 0,C 180,E1 -28536.401,E2 -28536.401} C_VEL
LIN {X 0,Y 66.717,Z 716.077,A -85,B 0,C 180,E1 -28545.275,E2 -28545.275} C_VEL
LIN {X 0,Y 68.08,Z 710.939,A -85,B 0,C 180,E1 -28554.395,E2 -28554.395} C_VEL
LIN {X 0,Y 70.286,Z 705.608,A -85,B 0,C 180,E1 -28561.671,E2 -28561.671} C_VEL
LIN {X 0,Y 73.408,Z 697.361,A -85,B 0,C 180,E1 -28570.424,E2 -28570.424} C_VEL
LIN {X 0,Y 76.879,Z 689.166,A -85,B 0,C 180,E1 -28577.005,E2 -28577.005} C_VEL
LIN {X 0,Y 81.019,Z 679.126,A -85,B 0,C 180,E1 -28583.156,E2 -28583.156} C_VEL
LIN {X 0,Y 84.995,Z 668.161,A -85,B 0,C 180,E1 -28588.362,E2 -28588.362} C_VEL
LIN {X 0,Y 86.897,Z 661.817,A -85,B 0,C 180,E1 -28590.968,E2 -28590.968} C_VEL
LIN {X 0,Y 86.923,Z 658.69,A -85,B 0,C 180,E1 -28592.805,E2 -28592.805} C_VEL
LIN {X 0,Y 86.188,Z 652.408,A -85,B 0,C 180,E1 -28597.21,E2 -28597.21} C_VEL
LIN {X 0,Y 85.02,Z 646.407,A -85,B 0,C 180,E1 -28602.207,E2 -28602.207} C_VEL
LIN {X 0,Y 84.298,Z 642.922,A -85,B 0,C 180,E1 -28605.514,E2 -28605.514} C_VEL
LIN {X 0,Y 83.13,Z 638.987,A -85,B 0,C 180,E1 -28610.264,E2 -28610.264} C_VEL
LIN {X 0,Y 81.09,Z 634.632,A -85,B 0,C 180,E1 -28619.998,E2 -28619.998} C_VEL
LIN {X 0,Y 80.47,Z 633.738,A -85,B 0,C 180,E1 -28625.008,E2 -28625.008} C_VEL
LIN {X 0,Y 80.137,Z 633.703,A -85,B 0,C 180,E1 -28630.1,E2 -28630.1} C_VEL
LIN {X 0,Y 80.179,Z 634.385,A -85,B 0,C 180,E1 -28635.362,E2 -28635.362} C_VEL
LIN {X 0,Y 81.709,Z 638.977,A -85,B 0,C 180,E1 -28648.231,E2 -28648.231} C_VEL
LIN {X 0,Y 82.869,Z 641.792,A -85,B 0,C 180,E1 -28653.448,E2 -28653.448} C_VEL
LIN {X 0,Y 84.911,Z 647.628,A -85,B 0,C 180,E1 -28661.462,E2 -28661.462} C_VEL
LIN {X 0,Y 86.181,Z 652.987,A -85,B 0,C 180,E1 -28667.215,E2 -28667.215} C_VEL
LIN {X 0,Y 86.964,Z 657.708,A -85,B 0,C 180,E1 -28671.728,E2 -28671.728} C_VEL
LIN {X 0,Y 87.295,Z 663.953,A -85,B 0,C 180,E1 -28677.194,E2 -28677.194} C_VEL
LIN {X 0,Y 86.87,Z 665.811,A -85,B 0,C 180,E1 -28678.499,E2 -28678.499} C_VEL
LIN {X 0,Y 82.091,Z 674.139,A -85,B 0,C 180,E1 -28683.286,E2 -28683.286} C_VEL
LIN {X 0,Y 76.817,Z 682.586,A -85,B 0,C 180,E1 -28689.93,E2 -28689.93} C_VEL
LIN {X 0,Y 74.035,Z 686.834,A -85,B 0,C 180,E1 -28694.244,E2 -28694.244} C_VEL
LIN {X 0,Y 71.439,Z 689.947,A -85,B 0,C 180,E1 -28697.641,E2 -28697.641} C_VEL
LIN {X 0,Y 66.079,Z 694.632,A -85,B 0,C 180,E1 -28703.41,E2 -28703.41} C_VEL
LIN {X 0,Y 61.372,Z 698.707,A -85,B 0,C 180,E1 -28710.392,E2 -28710.392} C_VEL
LIN {X 0,Y 59.965,Z 700.768,A -85,B 0,C 180,E1 -28715.451,E2 -28715.451} C_VEL
LIN {X 0,Y 59.686,Z 703.347,A -85,B 0,C 180,E1 -28723.615,E2 -28723.615} C_VEL
LIN {X 0,Y 60.512,Z 705.321,A -85,B 0,C 180,E1 -28731.708,E2 -28731.708} C_VEL
LIN {X 0,Y 63.737,Z 707.157,A -85,B 0,C 180,E1 -28743.451,E2 -28743.451} C_VEL
LIN {X 0,Y 66.479,Z 707.606,A -85,B 0,C 180,E1 -28749.361,E2 -28749.361} C_VEL
LIN {X 0,Y 66.612,Z 707.894,A -85,B 0,C 180,E1 -28752.396,E2 -28752.396} C_VEL
LIN {X 0,Y 60.522,Z 709.622,A -85,B 0,C 180,E1 -28764.509,E2 -28764.509} C_VEL
LIN {X 0,Y 58.145,Z 711.386,A -85,B 0,C 180,E1 -28782.939,E2 -28782.939} C_VEL
LIN {X 0,Y 58.166,Z 720.283,A -85,B 0,C 180,E1 -28793.063,E2 -28793.063} C_VEL
LIN {X 0,Y 59.614,Z 727.97,A -85,B 0,C 180,E1 -28803.382,E2 -28803.382} C_VEL
LIN {X 0,Y 64.125,Z 736.264,A -85,B 0,C 180,E1 -28815.905,E2 -28815.905} C_VEL
LIN {X 0,Y 70.578,Z 742.522,A -85,B 0,C 180,E1 -28825.538,E2 -28825.538} C_VEL
LIN {X 0,Y 80.591,Z 748.56,A -85,B 0,C 180,E1 -28834.532,E2 -28834.532} C_VEL
LIN {X 0,Y 83.191,Z 749.747,A -85,B 0,C 180,E1 -28836.256,E2 -28836.256} C_VEL
LIN {X 0,Y 81.018,Z 749.213,A -85,B 0,C 180,E1 -28838.682,E2 -28838.682} C_VEL
LIN {X 0,Y 70.208,Z 744.607,A -85,B 0,C 180,E1 -28849.415,E2 -28849.415} C_VEL
LIN {X 0,Y 63.329,Z 738.417,A -85,B 0,C 180,E1 -28863.653,E2 -28863.653} C_VEL
LIN {X 0,Y 61.57,Z 731.98,A -85,B 0,C 180,E1 -28876.81,E2 -28876.81} C_VEL
LIN {X 0,Y 61.567,Z 729.091,A -85,B 0,C 180,E1 -28881.803,E2 -28881.803} C_VEL
LIN {X 0,Y 61.051,Z 725.391,A -85,B 0,C 180,E1 -28886.706,E2 -28886.706} C_VEL
LIN {X 0,Y 60.47,Z 720.021,A -85,B 0,C 180,E1 -28892.921,E2 -28892.921} C_VEL
LIN {X 0,Y 59.593,Z 716.196,A -85,B 0,C 180,E1 -28903.649,E2 -28903.649} C_VEL
LIN {X 0,Y 61.101,Z 710.516,A -85,B 0,C 180,E1 -28915.377,E2 -28915.377} C_VEL
LIN {X 0,Y 63.516,Z 705.186,A -85,B 0,C 180,E1 -28923.597,E2 -28923.597} C_VEL
LIN {X 0,Y 66.857,Z 697.551,A -85,B 0,C 180,E1 -28932.619,E2 -28932.619} C_VEL
LIN {X 0,Y 70.979,Z 689.014,A -85,B 0,C 180,E1 -28940.125,E2 -28940.125} C_VEL
LIN {X 0,Y 74.976,Z 680.552,A -85,B 0,C 180,E1 -28945.774,E2 -28945.774} C_VEL
LIN {X 0,Y 79.304,Z 670.402,A -85,B 0,C 180,E1 -28951.069,E2 -28951.069} C_VEL
LIN {X 0,Y 81.377,Z 664.773,A -85,B 0,C 180,E1 -28953.573,E2 -28953.573} C_VEL
LIN {X 0,Y 81.745,Z 662.939,A -85,B 0,C 180,E1 -28954.538,E2 -28954.538} C_VEL
LIN {X 0,Y 81.429,Z 656.155,A -85,B 0,C 180,E1 -28959.802,E2 -28959.802} C_VEL
LIN {X 0,Y 80.765,Z 650.705,A -85,B 0,C 180,E1 -28964.865,E2 -28964.865} C_VEL
LIN {X 0,Y 80.472,Z 648.252,A -85,B 0,C 180,E1 -28967.387,E2 -28967.387} C_VEL
LIN {X 0,Y 79.582,Z 644.616,A -85,B 0,C 180,E1 -28972.386,E2 -28972.386} C_VEL
LIN {X 0,Y 78.275,Z 641.502,A -85,B 0,C 180,E1 -28979.998,E2 -28979.998} C_VEL
LIN {X 0,Y 77.716,Z 640.3,A -85,B 0,C 180,E1 -28985.831,E2 -28985.831} C_VEL
LIN {X 0,Y 77.414,Z 640.333,A -85,B 0,C 180,E1 -28990.459,E2 -28990.459} C_VEL
LIN {X 0,Y 77.293,Z 641.286,A -85,B 0,C 180,E1 -28995.828,E2 -28995.828} C_VEL
LIN {X 0,Y 78.119,Z 644.809,A -85,B 0,C 180,E1 -29006.73,E2 -29006.73} C_VEL
LIN {X 0,Y 78.957,Z 647.502,A -85,B 0,C 180,E1 -29012.278,E2 -29012.278} C_VEL
LIN {X 0,Y 80.308,Z 652.596,A -85,B 0,C 180,E1 -29020.018,E2 -29020.018} C_VEL
LIN {X 0,Y 81.1,Z 657.73,A -85,B 0,C 180,E1 -29026.105,E2 -29026.105} C_VEL
LIN {X 0,Y 81.479,Z 662.822,A -85,B 0,C 180,E1 -29031.41,E2 -29031.41} C_VEL
LIN {X 0,Y 81.45,Z 665.997,A -85,B 0,C 180,E1 -29034.507,E2 -29034.507} C_VEL
LIN {X 0,Y 80.939,Z 667.845,A -85,B 0,C 180,E1 -29035.899,E2 -29035.899} C_VEL
LIN {X 0,Y 74.824,Z 677.466,A -85,B 0,C 180,E1 -29041.984,E2 -29041.984} C_VEL
LIN {X 0,Y 69.302,Z 685.511,A -85,B 0,C 180,E1 -29049.205,E2 -29049.205} C_VEL
LIN {X 0,Y 64.759,Z 692.073,A -85,B 0,C 180,E1 -29057.603,E2 -29057.603} C_VEL
LIN {X 0,Y 61.559,Z 697.177,A -85,B 0,C 180,E1 -29066.722,E2 -29066.722} C_VEL
LIN {X 0,Y 59.965,Z 700.768,A -85,B 0,C 180,E1 -29075.451,E2 -29075.451} C_VEL
LIN {X 0,Y 58.973,Z 702.639,A -85,B 0,C 180,E1 -29080.768,E2 -29080.768} C_VEL
LIN {X 0,Y 56.638,Z 705.276,A -85,B 0,C 180,E1 -29089.97,E2 -29089.97} C_VEL
LIN {X 0,Y 55.794,Z 707.319,A -85,B 0,C 180,E1 -29099.872,E2 -29099.872} C_VEL
LIN {X 0,Y 57.107,Z 708.052,A -85,B 0,C 180,E1 -29105.679,E2 -29105.679} C_VEL
LIN {X 0,Y 58.799,Z 708.459,A -85,B 0,C 180,E1 -29109.512,E2 -29109.512} C_VEL
LIN {X 0,Y 57.905,Z 708.949,A -85,B 0,C 180,E1 -29113.266,E2 -29113.266} C_VEL
LIN {X 0,Y 51.245,Z 711.739,A -85,B 0,C 180,E1 -29135.709,E2 -29135.709} C_VEL
LIN {X 0,Y 51.391,Z 712.883,A -85,B 0,C 180,E1 -29148.293,E2 -29148.293} C_VEL
LIN {X 0,Y 52.258,Z 721.652,A -85,B 0,C 180,E1 -29160.003,E2 -29160.003} C_VEL
LIN {X 0,Y 55.496,Z 730.061,A -85,B 0,C 180,E1 -29172.807,E2 -29172.807} C_VEL
LIN {X 0,Y 61.064,Z 737.062,A -85,B 0,C 180,E1 -29183.761,E2 -29183.761} C_VEL
LIN {X 0,Y 69.771,Z 743.705,A -85,B 0,C 180,E1 -29193.646,E2 -29193.646} C_VEL
LIN {X 0,Y 73.283,Z 745.734,A -85,B 0,C 180,E1 -29196.473,E2 -29196.473} C_VEL
LIN {X 0,Y 71.98,Z 745.333,A -85,B 0,C 180,E1 -29198.647,E2 -29198.647} C_VEL
LIN {X 0,Y 63.386,Z 740.967,A -85,B 0,C 180,E1 -29208.306,E2 -29208.306} C_VEL
LIN {X 0,Y 57.605,Z 735.523,A -85,B 0,C 180,E1 -29220.798,E2 -29220.798} C_VEL
LIN {X 0,Y 55.397,Z 728.813,A -85,B 0,C 180,E1 -29235.309,E2 -29235.309} C_VEL
LIN {X 0,Y 55.231,Z 725.672,A -85,B 0,C 180,E1 -29240.855,E2 -29240.855} C_VEL
LIN {X 0,Y 54.151,Z 719.963,A -85,B 0,C 180,E1 -29248.612,E2 -29248.612} C_VEL
LIN {X 0,Y 52.529,Z 716.187,A -85,B 0,C 180,E1 -29261.584,E2 -29261.584} C_VEL
LIN {X 0,Y 53.419,Z 711.655,A -85,B 0,C 180,E1 -29273.254,E2 -29273.254} C_VEL
LIN {X 0,Y 56.356,Z 705.878,A -85,B 0,C 180,E1 -29284.145,E2 -29284.145} C_VEL
LIN {X 0,Y 60.097,Z 698.365,A -85,B 0,C 180,E1 -29294.569,E2 -29294.569} C_VEL
LIN {X 0,Y 64.365,Z 690.633,A -85,B 0,C 180,E1 -29302.346,E2 -29302.346} C_VEL
LIN {X 0,Y 69.435,Z 681.277,A -85,B 0,C 180,E1 -29309.226,E2 -29309.226} C_VEL
LIN {X 0,Y 74.6,Z 670.632,A -85,B 0,C 180,E1 -29315.072,E2 -29315.072} C_VEL
LIN {X 0,Y 76.35,Z 666.503,A -85,B 0,C 180,E1 -29317.01,E2 -29317.01} C_VEL
LIN {X 0,Y 76.644,Z 664.5,A -85,B 0,C 180,E1 -29318.48,E2 -29318.48} C_VEL
LIN {X 0,Y 76.681,Z 658.381,A -85,B 0,C 180,E1 -29324.038,E2 -29324.038} C_VEL
LIN {X 0,Y 76.439,Z 653.414,A -85,B 0,C 180,E1 -29329.402,E2 -29329.402} C_VEL
LIN {X 0,Y 76.172,Z 651.586,A -85,B 0,C 180,E1 -29332.043,E2 -29332.043} C_VEL
LIN {X 0,Y 75.809,Z 650.149,A -85,B 0,C 180,E1 -29334.679,E2 -29334.679} C_VEL
LIN {X 0,Y 75.119,Z 648.112,A -85,B 0,C 180,E1 -29339.998,E2 -29339.998} C_VEL
LIN {X 0,Y 74.754,Z 646.734,A -85,B 0,C 180,E1 -29345.392,E2 -29345.392} C_VEL
LIN {X 0,Y 74.293,Z 646.887,A -85,B 0,C 180,E1 -29350.904,E2 -29350.904} C_VEL
LIN {X 0,Y 73.934,Z 648.458,A -85,B 0,C 180,E1 -29358.075,E2 -29358.075} C_VEL
LIN {X 0,Y 74.329,Z 650.516,A -85,B 0,C 180,E1 -29365.116,E2 -29365.116} C_VEL
LIN {X 0,Y 74.863,Z 653.079,A -85,B 0,C 180,E1 -29371.087,E2 -29371.087} C_VEL
LIN {X 0,Y 75.521,Z 656.971,A -85,B 0,C 180,E1 -29377.745,E2 -29377.745} C_VEL
LIN {X 0,Y 75.88,Z 661.648,A -85,B 0,C 180,E1 -29383.993,E2 -29383.993} C_VEL
LIN {X 0,Y 75.875,Z 666.382,A -85,B 0,C 180,E1 -29389.574,E2 -29389.574} C_VEL
LIN {X 0,Y 75.72,Z 668.508,A -85,B 0,C 180,E1 -29391.86,E2 -29391.86} C_VEL
LIN {X 0,Y 75.174,Z 669.831,A -85,B 0,C 180,E1 -29392.915,E2 -29392.915} C_VEL
LIN {X 0,Y 68.66,Z 679.253,A -85,B 0,C 180,E1 -29399.21,E2 -29399.21} C_VEL
LIN {X 0,Y 62.709,Z 687.148,A -85,B 0,C 180,E1 -29406.899,E2 -29406.899} C_VEL
LIN {X 0,Y 57.865,Z 693.488,A -85,B 0,C 180,E1 -29415.935,E2 -29415.935} C_VEL
LIN {X 0,Y 54.4,Z 698.58,A -85,B 0,C 180,E1 -29426.29,E2 -29426.29} C_VEL
LIN {X 0,Y 52.709,Z 702.551,A -85,B 0,C 180,E1 -29437.655,E2 -29437.655} C_VEL
LIN {X 0,Y 52.725,Z 704.614,A -85,B 0,C 180,E1 -29445.454,E2 -29445.454} C_VEL
LIN {X 0,Y 53.724,Z 706.365,A -85,B 0,C 180,E1 -29453.699,E2 -29453.699} C_VEL
LIN {X 0,Y 57.107,Z 708.052,A -85,B 0,C 180,E1 -29465.679,E2 -29465.679} C_VEL
LIN {X 0,Y 57.471,Z 708.482,A -85,B 0,C 180,E1 -29468.711,E2 -29468.711} C_VEL
LIN {X 0,Y 56.384,Z 709.139,A -85,B 0,C 180,E1 -29472.62,E2 -29472.62} C_VEL
LIN {X 0,Y 53.419,Z 710.052,A -85,B 0,C 180,E1 -29477.844,E2 -29477.844} C_VEL
LIN {X 0,Y 44.843,Z 712.166,A -85,B 0,C 180,E1 -29493.212,E2 -29493.212} C_VEL
LIN {X 0,Y 43.956,Z 712.743,A -85,B 0,C 180,E1 -29498.934,E2 -29498.934} C_VEL
LIN {X 0,Y 45.16,Z 714.323,A -85,B 0,C 180,E1 -29515.541,E2 -29515.541} C_VEL
LIN {X 0,Y 47.22,Z 722.754,A -85,B 0,C 180,E1 -29528.563,E2 -29528.563} C_VEL
LIN {X 0,Y 52.11,Z 730.895,A -85,B 0,C 180,E1 -29541.774,E2 -29541.774} C_VEL
LIN {X 0,Y 61.606,Z 739.51,A -85,B 0,C 180,E1 -29554.781,E2 -29554.781} C_VEL
LIN {X 0,Y 64.079,Z 741.121,A -85,B 0,C 180,E1 -29557.046,E2 -29557.046} C_VEL
LIN {X 0,Y 63.034,Z 740.655,A -85,B 0,C 180,E1 -29558.707,E2 -29558.707} C_VEL
LIN {X 0,Y 54.953,Z 735.497,A -85,B 0,C 180,E1 -29570.258,E2 -29570.258} C_VEL
LIN {X 0,Y 50.216,Z 729.122,A -85,B 0,C 180,E1 -29585.182,E2 -29585.182} C_VEL
LIN {X 0,Y 49.299,Z 724.441,A -85,B 0,C 180,E1 -29595.561,E2 -29595.561} C_VEL
LIN {X 0,Y 48.912,Z 722.02,A -85,B 0,C 180,E1 -29599.661,E2 -29599.661} C_VEL
LIN {X 0,Y 48.365,Z 719.893,A -85,B 0,C 180,E1 -29602.703,E2 -29602.703} C_VEL
LIN {X 0,Y 45.931,Z 717.307,A -85,B 0,C 180,E1 -29614.396,E2 -29614.396} C_VEL
LIN {X 0,Y 45.647,Z 713.441,A -85,B 0,C 180,E1 -29627.943,E2 -29627.943} C_VEL
LIN {X 0,Y 47.87,Z 708.419,A -85,B 0,C 180,E1 -29640.93,E2 -29640.93} C_VEL
LIN {X 0,Y 50.3,Z 704.293,A -85,B 0,C 180,E1 -29648.967,E2 -29648.967} C_VEL
LIN {X 0,Y 55.033,Z 696.461,A -85,B 0,C 180,E1 -29660.315,E2 -29660.315} C_VEL
LIN {X 0,Y 61.117,Z 686.935,A -85,B 0,C 180,E1 -29669.603,E2 -29669.603} C_VEL
LIN {X 0,Y 66.504,Z 677.915,A -85,B 0,C 180,E1 -29675.817,E2 -29675.817} C_VEL
LIN {X 0,Y 71.159,Z 669.085,A -85,B 0,C 180,E1 -29680.493,E2 -29680.493} C_VEL
LIN {X 0,Y 71.586,Z 667.934,A -85,B 0,C 180,E1 -29681.24,E2 -29681.24} C_VEL
LIN {X 0,Y 72.091,Z 662.135,A -85,B 0,C 180,E1 -29687.15,E2 -29687.15} C_VEL
LIN {X 0,Y 72.242,Z 658.39,A -85,B 0,C 180,E1 -29691.607,E2 -29691.607} C_VEL
LIN {X 0,Y 72.125,Z 656.683,A -85,B 0,C 180,E1 -29694.406,E2 -29694.406} C_VEL
LIN {X 0,Y 71.608,Z 654.509,A -85,B 0,C 180,E1 -29699.998,E2 -29699.998} C_VEL
LIN {X 0,Y 71.277,Z 653.005,A -85,B 0,C 180,E1 -29706.25,E2 -29706.25} C_VEL
LIN {X 0,Y 70.762,Z 653.305,A -85,B 0,C 180,E1 -29711.455,E2 -29711.455} C_VEL
LIN {X 0,Y 70.295,Z 654.541,A -85,B 0,C 180,E1 -29717.451,E2 -29717.451} C_VEL
LIN {X 0,Y 70.349,Z 656.155,A -85,B 0,C 180,E1 -29723.551,E2 -29723.551} C_VEL
LIN {X 0,Y 70.566,Z 658.548,A -85,B 0,C 180,E1 -29729.863,E2 -29729.863} C_VEL
LIN {X 0,Y 70.76,Z 662.103,A -85,B 0,C 180,E1 -29736.576,E2 -29736.576} C_VEL
LIN {X 0,Y 70.661,Z 666.102,A -85,B 0,C 180,E1 -29742.497,E2 -29742.497} C_VEL
LIN {X 0,Y 70.339,Z 669.68,A -85,B 0,C 180,E1 -29747.207,E2 -29747.207} C_VEL
LIN {X 0,Y 70.182,Z 670.719,A -85,B 0,C 180,E1 -29748.521,E2 -29748.521} C_VEL
LIN {X 0,Y 69.593,Z 671.907,A -85,B 0,C 180,E1 -29749.513,E2 -29749.513} C_VEL
LIN {X 0,Y 62.694,Z 681.036,A -85,B 0,C 180,E1 -29755.903,E2 -29755.903} C_VEL
LIN {X 0,Y 56.22,Z 688.755,A -85,B 0,C 180,E1 -29764.047,E2 -29764.047} C_VEL
LIN {X 0,Y 50.99,Z 694.981,A -85,B 0,C 180,E1 -29773.991,E2 -29773.991} C_VEL
LIN {X 0,Y 47.265,Z 699.98,A -85,B 0,C 180,E1 -29785.728,E2 -29785.728} C_VEL
LIN {X 0,Y 45.605,Z 703.861,A -85,B 0,C 180,E1 -29798.857,E2 -29798.857} C_VEL
LIN {X 0,Y 45.824,Z 705.886,A -85,B 0,C 180,E1 -29807.854,E2 -29807.854} C_VEL
LIN {X 0,Y 47.074,Z 707.459,A -85,B 0,C 180,E1 -29816.599,E2 -29816.599} C_VEL
LIN {X 0,Y 50.509,Z 709.024,A -85,B 0,C 180,E1 -29828.273,E2 -29828.273} C_VEL
LIN {X 0,Y 49.219,Z 709.874,A -85,B 0,C 180,E1 -29834.447,E2 -29834.447} C_VEL
LIN {X 0,Y 43.956,Z 712.743,A -85,B 0,C 180,E1 -29858.934,E2 -29858.934} C_VEL
LIN {X 0,Y 43.324,Z 713.342,A -85,B 0,C 180,E1 -29864.234,E2 -29864.234} C_VEL
LIN {X 0,Y 41.281,Z 714.29,A -85,B 0,C 180,E1 -29873.184,E2 -29873.184} C_VEL
LIN {X 0,Y 39.902,Z 715.513,A -85,B 0,C 180,E1 -29883.199,E2 -29883.199} C_VEL
LIN {X 0,Y 40.189,Z 716.922,A -85,B 0,C 180,E1 -29887.22,E2 -29887.22} C_VEL
LIN {X 0,Y 45.088,Z 726.082,A -85,B 0,C 180,E1 -29902.938,E2 -29902.938} C_VEL
LIN {X 0,Y 53.384,Z 734.382,A -85,B 0,C 180,E1 -29915.799,E2 -29915.799} C_VEL
LIN {X 0,Y 54.376,Z 735.273,A -85,B 0,C 180,E1 -29919.161,E2 -29919.161} C_VEL
LIN {X 0,Y 46.917,Z 729.253,A -85,B 0,C 180,E1 -29933.199,E2 -29933.199} C_VEL
LIN {X 0,Y 43.55,Z 721.827,A -85,B 0,C 180,E1 -29951.18,E2 -29951.18} C_VEL
LIN {X 0,Y 42.974,Z 719.662,A -85,B 0,C 180,E1 -29955.809,E2 -29955.809} C_VEL
LIN {X 0,Y 38.74,Z 716.014,A -85,B 0,C 180,E1 -29975.214,E2 -29975.214} C_VEL
LIN {X 0,Y 38.812,Z 712.056,A -85,B 0,C 180,E1 -29991.243,E2 -29991.243} C_VEL
LIN {X 0,Y 42.538,Z 705.984,A -85,B 0,C 180,E1 -30008.294,E2 -30008.294} C_VEL
LIN {X 0,Y 47.263,Z 699.086,A -85,B 0,C 180,E1 -30021.095,E2 -30021.095} C_VEL
LIN {X 0,Y 53.852,Z 690.189,A -85,B 0,C 180,E1 -30031.766,E2 -30031.766} C_VEL
LIN {X 0,Y 60.225,Z 681.119,A -85,B 0,C 180,E1 -30039.013,E2 -30039.013} C_VEL
LIN {X 0,Y 65.78,Z 672.279,A -85,B 0,C 180,E1 -30044.083,E2 -30044.083} C_VEL
LIN {X 0,Y 66.709,Z 670.438,A -85,B 0,C 180,E1 -30045.203,E2 -30045.203} C_VEL
LIN {X 0,Y 67.57,Z 665.465,A -85,B 0,C 180,E1 -30051.022,E2 -30051.022} C_VEL
